  MoveL (T13144) to (117.57, 104.7, 14.9) mm, rotated rx 180 ry 0 rz -180 deg; joints [0, 0, 0, 0, 0, 0]
  Call Extruder 0.0175
  MoveL (T13145) to (117.21, 105.06, 14.9) mm, rotated rx 180 ry 0 rz -180 deg; joints [0, 0, 0, 0, 0, 0]
  Call Extruder 0.02231
  MoveL (T13146) to (117.21, 104.41, 14.9) mm, rotated rx 180 ry 0 rz -180 deg; joints [0, 0, 0, 0, 0, 0]
  Call Extruder 0.0264
  MoveL (T13147) to (117.75, 103.87, 14.9) mm, rotated rx 180 ry 0 rz -180 deg; joints [0, 0, 0, 0, 0, 0]
  Set speed (45.0 mm/s)
  Call Extruder -1.6
  MoveL (T13148) to (117.75, 103.87, 14.9) mm, rotated rx 180 ry 0 rz -180 deg; joints [0, 0, 0, 0, 0, 0]
  Set speed (120.0 mm/s)
  MoveL (T13149) to (117.75, 103.87, 14.9) mm, rotated rx 180 ry 0 rz -180 deg; joints [0, 0, 0, 0, 0, 0]
  Call Extruder -0.27367
  MoveL (T13150) to (117.21, 104.41, 14.9) mm, rotated rx 180 ry 0 rz -180 deg; joints [0, 0, 0, 0, 0, 0]
  Call Extruder -0.10633
  MoveL (T13151) to (117.21, 104.71, 14.9) mm, rotated rx 180 ry 0 rz -180 deg; joints [0, 0, 0, 0, 0, 0]
  Set speed (45.0 mm/s)
  Call Extruder -0.02
  MoveL (T13152) to (117.21, 104.71, 14.9) mm, rotated rx 180 ry 0 rz -180 deg; joints [0, 0, 0, 0, 0, 0]
  Set speed (150.0 mm/s)
  MoveL (T13153) to (117.21, 104.71, 16.9) mm, rotated rx 180 ry 0 rz -180 deg; joints [0, 0, 0, 0, 0, 0]
  MoveL (T13154) to (121.1, 106.08, 16.9) mm, rotated rx 180 ry 0 rz -180 deg; joints [0, 0, 0, 0, 0, 0]
  MoveL (T13155) to (121.1, 106.08, 14.9) mm, rotated rx 180 ry 0 rz -180 deg; joints [0, 0, 0, 0, 0, 0]
  Set speed (40.0 mm/s)
  Call Extruder 2.0
  MoveL (T13156) to (121.1, 106.08, 14.9) mm, rotated rx 180 ry 0 rz -180 deg; joints [0, 0, 0, 0, 0, 0]
  Set speed (28.1 mm/s)
  MoveL (T13157) to (121.1, 106.08, 14.9) mm, rotated rx 180 ry 0 rz -180 deg; joints [0, 0, 0, 0, 0, 0]
  Call Extruder 0.02425
  MoveL (T13158) to (120.59, 106.58, 14.9) mm, rotated rx 180 ry 0 rz -180 deg; joints [0, 0, 0, 0, 0, 0]
  Call Extruder 0.02201
  MoveL (T13159) to (119.95, 106.58, 14.9) mm, rotated rx 180 ry 0 rz -180 deg; joints [0, 0, 0, 0, 0, 0]
  Call Extruder 0.01541
  MoveL (T13160) to (120.27, 106.27, 14.9) mm, rotated rx 180 ry 0 rz -180 deg; joints [0, 0, 0, 0, 0, 0]
  Call Extruder 0.02201
  MoveL (T13161) to (119.62, 106.27, 14.9) mm, rotated rx 180 ry 0 rz -180 deg; joints [0, 0, 0, 0, 0, 0]
  Call Extruder 0.01442
  MoveL (T13162) to (119.33, 106.56, 14.9) mm, rotated rx 180 ry 0 rz -180 deg; joints [0, 0, 0, 0, 0, 0]
  Set speed (45.0 mm/s)
  Call Extruder -1.6
  MoveL (T13163) to (119.33, 106.56, 14.9) mm, rotated rx 180 ry 0 rz -180 deg; joints [0, 0, 0, 0, 0, 0]
  Set speed (120.0 mm/s)
  MoveL (T13164) to (119.33, 106.56, 14.9) mm, rotated rx 180 ry 0 rz -180 deg; joints [0, 0, 0, 0, 0, 0]
  Call Extruder -0.1506
  MoveL (T13165) to (119.62, 106.27, 14.9) mm, rotated rx 180 ry 0 rz -180 deg; joints [0, 0, 0, 0, 0, 0]
  Call Extruder -0.2294
  MoveL (T13166) to (120.27, 106.27, 14.9) mm, rotated rx 180 ry 0 rz -180 deg; joints [0, 0, 0, 0, 0, 0]
  Set speed (45.0 mm/s)
  Call Extruder -0.02
  MoveL (T13167) to (120.27, 106.27, 14.9) mm, rotated rx 180 ry 0 rz -180 deg; joints [0, 0, 0, 0, 0, 0]
  Set speed (150.0 mm/s)
  MoveL (T13168) to (120.27, 106.27, 16.9) mm, rotated rx 180 ry 0 rz -180 deg; joints [0, 0, 0, 0, 0, 0]
  MoveL (T13169) to (119.17, 110.71, 16.9) mm, rotated rx 180 ry 0 rz -180 deg; joints [0, 0, 0, 0, 0, 0]
  MoveL (T13170) to (119.17, 110.71, 14.9) mm, rotated rx 180 ry 0 rz -180 deg; joints [0, 0, 0, 0, 0, 0]
  Set speed (40.0 mm/s)
  Call Extruder 2.0
  MoveL (T13171) to (119.17, 110.71, 14.9) mm, rotated rx 180 ry 0 rz -180 deg; joints [0, 0, 0, 0, 0, 0]
  Set speed (28.1 mm/s)
  MoveL (T13172) to (119.17, 110.71, 14.9) mm, rotated rx 180 ry 0 rz -180 deg; joints [0, 0, 0, 0, 0, 0]
  Call Extruder 0.0033
  MoveL (T13173) to (119.1, 110.78, 14.9) mm, rotated rx 180 ry 0 rz -180 deg; joints [0, 0, 0, 0, 0, 0]
  Call Extruder 0.015
  MoveL (T13174) to (119.1, 111.28, 14.9) mm, rotated rx 180 ry 0 rz -180 deg; joints [0, 0, 0, 0, 0, 0]
  Call Extruder 0.01378
  MoveL (T13175) to (119.42, 111.6, 14.9) mm, rotated rx 180 ry 0 rz -180 deg; joints [0, 0, 0, 0, 0, 0]
  Call Extruder 0.04234
  MoveL (T13176) to (120.81, 111.6, 14.9) mm, rotated rx 180 ry 0 rz -180 deg; joints [0, 0, 0, 0, 0, 0]
  Call Extruder 0.01501
  MoveL (T13177) to (121.16, 111.94, 14.9) mm, rotated rx 180 ry 0 rz -180 deg; joints [0, 0, 0, 0, 0, 0]
  Call Extruder 0.01633
  MoveL (T13178) to (121.16, 112.48, 14.9) mm, rotated rx 180 ry 0 rz -180 deg; joints [0, 0, 0, 0, 0, 0]
  Call Extruder 0.05296
  MoveL (T13179) to (119.42, 112.48, 14.9) mm, rotated rx 180 ry 0 rz -180 deg; joints [0, 0, 0, 0, 0, 0]
  Call Extruder 0.00512
  MoveL (T13180) to (119.3, 112.6, 14.9) mm, rotated rx 180 ry 0 rz -180 deg; joints [0, 0, 0, 0, 0, 0]
  Set speed (150.0 mm/s)
  MoveL (T13181) to (121, 112.7, 14.9) mm, rotated rx 180 ry 0 rz -180 deg; joints [0, 0, 0, 0, 0, 0]
  Set speed (28.1 mm/s)
  MoveL (T13182) to (121, 112.7, 14.9) mm, rotated rx 180 ry 0 rz -180 deg; joints [0, 0, 0, 0, 0, 0]
  Call Extruder 0.01588
  MoveL (T13183) to (120.65, 113.05, 14.9) mm, rotated rx 180 ry 0 rz -180 deg; joints [0, 0, 0, 0, 0, 0]
  Call Extruder 0.01956
  MoveL (T13184) to (120.04, 113.05, 14.9) mm, rotated rx 180 ry 0 rz -180 deg; joints [0, 0, 0, 0, 0, 0]
  Call Extruder 0.00755
  MoveL (T13185) to (120.21, 112.89, 14.9) mm, rotated rx 180 ry 0 rz -180 deg; joints [0, 0, 0, 0, 0, 0]
  Call Extruder 0.01956
  MoveL (T13186) to (119.6, 112.89, 14.9) mm, rotated rx 180 ry 0 rz -180 deg; joints [0, 0, 0, 0, 0, 0]
  Call Extruder 0.01277
  MoveL (T13187) to (119.32, 113.17, 14.9) mm, rotated rx 180 ry 0 rz -180 deg; joints [0, 0, 0, 0, 0, 0]
  Set speed (45.0 mm/s)
  Call Extruder -1.6
  MoveL (T13188) to (119.32, 113.17, 14.9) mm, rotated rx 180 ry 0 rz -180 deg; joints [0, 0, 0, 0, 0, 0]
  Set speed (120.0 mm/s)
  MoveL (T13189) to (119.32, 113.17, 14.9) mm, rotated rx 180 ry 0 rz -180 deg; joints [0, 0, 0, 0, 0, 0]
  Call Extruder -0.14132
  MoveL (T13190) to (119.6, 112.89, 14.9) mm, rotated rx 180 ry 0 rz -180 deg; joints [0, 0, 0, 0, 0, 0]
  Call Extruder -0.21648
  MoveL (T13191) to (120.21, 112.89, 14.9) mm, rotated rx 180 ry 0 rz -180 deg; joints [0, 0, 0, 0, 0, 0]
  Call Extruder -0.0222
  MoveL (T13192) to (120.17, 112.93, 14.9) mm, rotated rx 180 ry 0 rz -180 deg; joints [0, 0, 0, 0, 0, 0]
  Set speed (45.0 mm/s)
  Call Extruder -0.02
  MoveL (T13193) to (120.17, 112.93, 14.9) mm, rotated rx 180 ry 0 rz -180 deg; joints [0, 0, 0, 0, 0, 0]
  Set speed (150.0 mm/s)
  MoveL (T13194) to (120.17, 112.93, 16.9) mm, rotated rx 180 ry 0 rz -180 deg; joints [0, 0, 0, 0, 0, 0]
  MoveL (T13195) to (120.92, 110.82, 16.9) mm, rotated rx 180 ry 0 rz -180 deg; joints [0, 0, 0, 0, 0, 0]
  MoveL (T13196) to (120.92, 110.82, 14.9) mm, rotated rx 180 ry 0 rz -180 deg; joints [0, 0, 0, 0, 0, 0]
  Set speed (40.0 mm/s)
  Call Extruder 2.0
  MoveL (T13197) to (120.92, 110.82, 14.9) mm, rotated rx 180 ry 0 rz -180 deg; joints [0, 0, 0, 0, 0, 0]
  Set speed (28.1 mm/s)
  MoveL (T13198) to (120.92, 110.82, 14.9) mm, rotated rx 180 ry 0 rz -180 deg; joints [0, 0, 0, 0, 0, 0]
  Call Extruder 0.01748
  MoveL (T13199) to (120.55, 111.19, 14.9) mm, rotated rx 180 ry 0 rz -180 deg; joints [0, 0, 0, 0, 0, 0]
  Call Extruder 0.02083
  MoveL (T13200) to (119.92, 111.19, 14.9) mm, rotated rx 180 ry 0 rz -180 deg; joints [0, 0, 0, 0, 0, 0]
  Call Extruder 0.01748
  MoveL (T13201) to (120.29, 110.82, 14.9) mm, rotated rx 180 ry 0 rz -180 deg; joints [0, 0, 0, 0, 0, 0]
  Set speed (45.0 mm/s)
  Call Extruder -1.6
  MoveL (T13202) to (120.29, 110.82, 14.9) mm, rotated rx 180 ry 0 rz -180 deg; joints [0, 0, 0, 0, 0, 0]
  Set speed (120.0 mm/s)
  MoveL (T13203) to (120.29, 110.82, 14.9) mm, rotated rx 180 ry 0 rz -180 deg; joints [0, 0, 0, 0, 0, 0]
  Call Extruder -0.18757
  MoveL (T13204) to (119.92, 111.19, 14.9) mm, rotated rx 180 ry 0 rz -180 deg; joints [0, 0, 0, 0, 0, 0]
  Call Extruder -0.19243
  MoveL (T13205) to (120.46, 111.19, 14.9) mm, rotated rx 180 ry 0 rz -180 deg; joints [0, 0, 0, 0, 0, 0]
  Set speed (45.0 mm/s)
  Call Extruder -0.02
  MoveL (T13206) to (120.46, 111.19, 14.9) mm, rotated rx 180 ry 0 rz -180 deg; joints [0, 0, 0, 0, 0, 0]
  Set speed (150.0 mm/s)
  MoveL (T13207) to (120.46, 111.19, 16.9) mm, rotated rx 180 ry 0 rz -180 deg; joints [0, 0, 0, 0, 0, 0]
  MoveL (T13208) to (121.34, 117.66, 16.9) mm, rotated rx 180 ry 0 rz -180 deg; joints [0, 0, 0, 0, 0, 0]
  MoveL (T13209) to (121.34, 117.66, 14.9) mm, rotated rx 180 ry 0 rz -180 deg; joints [0, 0, 0, 0, 0, 0]
  Set speed (40.0 mm/s)
  Call Extruder 2.0
  MoveL (T13210) to (121.34, 117.66, 14.9) mm, rotated rx 180 ry 0 rz -180 deg; joints [0, 0, 0, 0, 0, 0]
  Set speed (28.1 mm/s)
  MoveL (T13211) to (121.34, 117.66, 14.9) mm, rotated rx 180 ry 0 rz -180 deg; joints [0, 0, 0, 0, 0, 0]
  Call Extruder 0.00963
  MoveL (T13212) to (121.15, 117.85, 14.9) mm, rotated rx 180 ry 0 rz -180 deg; joints [0, 0, 0, 0, 0, 0]
  Call Extruder 0.02452
  MoveL (T13213) to (120.47, 117.85, 14.9) mm, rotated rx 180 ry 0 rz -180 deg; joints [0, 0, 0, 0, 0, 0]
  Call Extruder 0.02041
  MoveL (T13214) to (120.87, 117.45, 14.9) mm, rotated rx 180 ry 0 rz -180 deg; joints [0, 0, 0, 0, 0, 0]
  Call Extruder 0.02452
  MoveL (T13215) to (120.19, 117.45, 14.9) mm, rotated rx 180 ry 0 rz -180 deg; joints [0, 0, 0, 0, 0, 0]
  Call Extruder 0.02041
  MoveL (T13216) to (119.79, 117.85, 14.9) mm, rotated rx 180 ry 0 rz -180 deg; joints [0, 0, 0, 0, 0, 0]
  Call Extruder 0.00326
  MoveL (T13217) to (119.7, 117.85, 14.9) mm, rotated rx 180 ry 0 rz -180 deg; joints [0, 0, 0, 0, 0, 0]
  Call Extruder 0.00991
  MoveL (T13218) to (119.5, 117.65, 14.9) mm, rotated rx 180 ry 0 rz -180 deg; joints [0, 0, 0, 0, 0, 0]
  Call Extruder 0.00726
  MoveL (T13219) to (119.5, 117.45, 14.9) mm, rotated rx 180 ry 0 rz -180 deg; joints [0, 0, 0, 0, 0, 0]
  Call Extruder 0.00961
  MoveL (T13220) to (119.69, 117.26, 14.9) mm, rotated rx 180 ry 0 rz -180 deg; joints [0, 0, 0, 0, 0, 0]
  Set speed (45.0 mm/s)
  Call Extruder -1.6
  MoveL (T13221) to (119.69, 117.26, 14.9) mm, rotated rx 180 ry 0 rz -180 deg; joints [0, 0, 0, 0, 0, 0]
  Set speed (120.0 mm/s)
  MoveL (T13222) to (119.69, 117.26, 14.9) mm, rotated rx 180 ry 0 rz -180 deg; joints [0, 0, 0, 0, 0, 0]
  Call Extruder -0.09501
  MoveL (T13223) to (119.5, 117.45, 14.9) mm, rotated rx 180 ry 0 rz -180 deg; joints [0, 0, 0, 0, 0, 0]
  Call Extruder -0.07173
  MoveL (T13224) to (119.5, 117.65, 14.9) mm, rotated rx 180 ry 0 rz -180 deg; joints [0, 0, 0, 0, 0, 0]
  Call Extruder -0.09794
  MoveL (T13225) to (119.7, 117.85, 14.9) mm, rotated rx 180 ry 0 rz -180 deg; joints [0, 0, 0, 0, 0, 0]
  Call Extruder -0.03219
  MoveL (T13226) to (119.79, 117.85, 14.9) mm, rotated rx 180 ry 0 rz -180 deg; joints [0, 0, 0, 0, 0, 0]
  Call Extruder -0.08312
  MoveL (T13227) to (119.95, 117.68, 14.9) mm, rotated rx 180 ry 0 rz -180 deg; joints [0, 0, 0, 0, 0, 0]
  Set speed (45.0 mm/s)
  Call Extruder -0.02
  MoveL (T13228) to (119.95, 117.68, 14.9) mm, rotated rx 180 ry 0 rz -180 deg; joints [0, 0, 0, 0, 0, 0]
  Set speed (150.0 mm/s)
  MoveL (T13229) to (119.95, 117.68, 16.9) mm, rotated rx 180 ry 0 rz -180 deg; joints [0, 0, 0, 0, 0, 0]
  MoveL (T13230) to (104.34, 103.54, 16.9) mm, rotated rx 180 ry 0 rz -180 deg; joints [0, 0, 0, 0, 0, 0]
  MoveL (T13231) to (104.34, 103.54, 15.1) mm, rotated rx 180 ry 0 rz -180 deg; joints [0, 0, 0, 0, 0, 0]
  Set speed (40.0 mm/s)
  Call Extruder 2.0
  MoveL (T13232) to (104.34, 103.54, 15.1) mm, rotated rx 180 ry 0 rz -180 deg; joints [0, 0, 0, 0, 0, 0]
  Set speed (28.8 mm/s)
  MoveL (T13233) to (104.34, 103.54, 15.1) mm, rotated rx 180 ry 0 rz -180 deg; joints [0, 0, 0, 0, 0, 0]
  Call Extruder 0.08935
  MoveL (T13234) to (107.27, 103.54, 15.1) mm, rotated rx 180 ry 0 rz -180 deg; joints [0, 0, 0, 0, 0, 0]
  Call Extruder 0.05791
  MoveL (T13235) to (107.27, 105.44, 15.1) mm, rotated rx 180 ry 0 rz -180 deg; joints [0, 0, 0, 0, 0, 0]
  Call Extruder 0.11368
  MoveL (T13236) to (111, 105.44, 15.1) mm, rotated rx 180 ry 0 rz -180 deg; joints [0, 0, 0, 0, 0, 0]
  Call Extruder 0.05791
  MoveL (T13237) to (111, 103.54, 15.1) mm, rotated rx 180 ry 0 rz -180 deg; joints [0, 0, 0, 0, 0, 0]
  Call Extruder 0.07022
  MoveL (T13238) to (113.31, 103.54, 15.1) mm, rotated rx 180 ry 0 rz -180 deg; joints [0, 0, 0, 0, 0, 0]
  Call Extruder 0.05791
  MoveL (T13239) to (113.31, 105.44, 15.1) mm, rotated rx 180 ry 0 rz -180 deg; joints [0, 0, 0, 0, 0, 0]
  Call Extruder 0.11332
  MoveL (T13240) to (117.03, 105.44, 15.1) mm, rotated rx 180 ry 0 rz -180 deg; joints [0, 0, 0, 0, 0, 0]
  Call Extruder 0.0579
  MoveL (T13241) to (117.03, 103.54, 15.1) mm, rotated rx 180 ry 0 rz -180 deg; joints [0, 0, 0, 0, 0, 0]
  Call Extruder 0.13501
  MoveL (T13242) to (121.46, 103.54, 15.1) mm, rotated rx 180 ry 0 rz -180 deg; joints [0, 0, 0, 0, 0, 0]
  Call Extruder 0.09842
  MoveL (T13243) to (121.46, 106.77, 15.1) mm, rotated rx 180 ry 0 rz -180 deg; joints [0, 0, 0, 0, 0, 0]
  Call Extruder 0.05868
  MoveL (T13244) to (119.53, 106.77, 15.1) mm, rotated rx 180 ry 0 rz -180 deg; joints [0, 0, 0, 0, 0, 0]
  Call Extruder 0.11599
  MoveL (T13245) to (119.53, 110.58, 15.1) mm, rotated rx 180 ry 0 rz -180 deg; joints [0, 0, 0, 0, 0, 0]
  Call Extruder 0.05873
  MoveL (T13246) to (121.46, 110.58, 15.1) mm, rotated rx 180 ry 0 rz -180 deg; joints [0, 0, 0, 0, 0, 0]
  Call Extruder 0.08813
  MoveL (T13247) to (121.46, 113.47, 15.1) mm, rotated rx 180 ry 0 rz -180 deg; joints [0, 0, 0, 0, 0, 0]
  Call Extruder 0.05877
  MoveL (T13248) to (119.53, 113.47, 15.1) mm, rotated rx 180 ry 0 rz -180 deg; joints [0, 0, 0, 0, 0, 0]
  Call Extruder 0.11538
  MoveL (T13249) to (119.53, 117.25, 15.1) mm, rotated rx 180 ry 0 rz -180 deg; joints [0, 0, 0, 0, 0, 0]
  Call Extruder 0.05882
  MoveL (T13250) to (121.46, 117.26, 15.1) mm, rotated rx 180 ry 0 rz -180 deg; joints [0, 0, 0, 0, 0, 0]
  Call Extruder 0.12804
  MoveL (T13251) to (121.46, 121.46, 15.1) mm, rotated rx 180 ry 0 rz -180 deg; joints [0, 0, 0, 0, 0, 0]
  Call Extruder 0.54596
  MoveL (T13252) to (103.54, 121.46, 15.1) mm, rotated rx 180 ry 0 rz -180 deg; joints [0, 0, 0, 0, 0, 0]
  Call Extruder 0.54596
  MoveL (T13253) to (103.54, 103.54, 15.1) mm, rotated rx 180 ry 0 rz -180 deg; joints [0, 0, 0, 0, 0, 0]
  Call Extruder 0.02254
  MoveL (T13254) to (104.28, 103.54, 15.1) mm, rotated rx 180 ry 0 rz -180 deg; joints [0, 0, 0, 0, 0, 0]
  Set speed (150.0 mm/s)
  MoveL (T13255) to (103.53, 103.13, 15.1) mm, rotated rx 180 ry 0 rz -180 deg; joints [0, 0, 0, 0, 0, 0]
  Set speed (28.8 mm/s)
  MoveL (T13256) to (103.53, 103.13, 15.1) mm, rotated rx 180 ry 0 rz -180 deg; joints [0, 0, 0, 0, 0, 0]
  Call Extruder 0.12635
  MoveL (T13257) to (107.68, 103.13, 15.1) mm, rotated rx 180 ry 0 rz -180 deg; joints [0, 0, 0, 0, 0, 0]
  Call Extruder 0.05791
  MoveL (T13258) to (107.68, 105.03, 15.1) mm, rotated rx 180 ry 0 rz -180 deg; joints [0, 0, 0, 0, 0, 0]
  Call Extruder 0.08888
  MoveL (T13259) to (110.6, 105.03, 15.1) mm, rotated rx 180 ry 0 rz -180 deg; joints [0, 0, 0, 0, 0, 0]
  Call Extruder 0.05791
  MoveL (T13260) to (110.6, 103.13, 15.1) mm, rotated rx 180 ry 0 rz -180 deg; joints [0, 0, 0, 0, 0, 0]
  Call Extruder 0.09501
  MoveL (T13261) to (113.72, 103.13, 15.1) mm, rotated rx 180 ry 0 rz -180 deg; joints [0, 0, 0, 0, 0, 0]
  Call Extruder 0.05791
  MoveL (T13262) to (113.72, 105.03, 15.1) mm, rotated rx 180 ry 0 rz -180 deg; joints [0, 0, 0, 0, 0, 0]
  Call Extruder 0.08852
  MoveL (T13263) to (116.62, 105.03, 15.1) mm, rotated rx 180 ry 0 rz -180 deg; joints [0, 0, 0, 0, 0, 0]
  Call Extruder 0.0579
  MoveL (T13264) to (116.62, 103.13, 15.1) mm, rotated rx 180 ry 0 rz -180 deg; joints [0, 0, 0, 0, 0, 0]
  Call Extruder 0.15982
  MoveL (T13265) to (121.87, 103.13, 15.1) mm, rotated rx 180 ry 0 rz -180 deg; joints [0, 0, 0, 0, 0, 0]
  Call Extruder 0.12322
  MoveL (T13266) to (121.87, 107.18, 15.1) mm, rotated rx 180 ry 0 rz -180 deg; joints [0, 0, 0, 0, 0, 0]
  Call Extruder 0.05868
  MoveL (T13267) to (119.94, 107.18, 15.1) mm, rotated rx 180 ry 0 rz -180 deg; joints [0, 0, 0, 0, 0, 0]
  Call Extruder 0.09119
  MoveL (T13268) to (119.94, 110.17, 15.1) mm, rotated rx 180 ry 0 rz -180 deg; joints [0, 0, 0, 0, 0, 0]
  Call Extruder 0.05872
  MoveL (T13269) to (121.87, 110.17, 15.1) mm, rotated rx 180 ry 0 rz -180 deg; joints [0, 0, 0, 0, 0, 0]
  Call Extruder 0.11295
  MoveL (T13270) to (121.87, 113.88, 15.1) mm, rotated rx 180 ry 0 rz -180 deg; joints [0, 0, 0, 0, 0, 0]
  Call Extruder 0.05877
  MoveL (T13271) to (119.94, 113.88, 15.1) mm, rotated rx 180 ry 0 rz -180 deg; joints [0, 0, 0, 0, 0, 0]
  Call Extruder 0.09058
  MoveL (T13272) to (119.94, 116.85, 15.1) mm, rotated rx 180 ry 0 rz -180 deg; joints [0, 0, 0, 0, 0, 0]
  Call Extruder 0.05881
  MoveL (T13273) to (121.87, 116.85, 15.1) mm, rotated rx 180 ry 0 rz -180 deg; joints [0, 0, 0, 0, 0, 0]
  Call Extruder 0.15282
  MoveL (T13274) to (121.87, 121.87, 15.1) mm, rotated rx 180 ry 0 rz -180 deg; joints [0, 0, 0, 0, 0, 0]
  Call Extruder 0.57077
  MoveL (T13275) to (103.13, 121.87, 15.1) mm, rotated rx 180 ry 0 rz -180 deg; joints [0, 0, 0, 0, 0, 0]
  Call Extruder 0.57077
  MoveL (T13276) to (103.13, 103.13, 15.1) mm, rotated rx 180 ry 0 rz -180 deg; joints [0, 0, 0, 0, 0, 0]
  Call Extruder 0.01036
  MoveL (T13277) to (103.47, 103.13, 15.1) mm, rotated rx 180 ry 0 rz -180 deg; joints [0, 0, 0, 0, 0, 0]
  Set speed (150.0 mm/s)
  MoveL (T13278) to (102.72, 102.81, 15.1) mm, rotated rx 180 ry 0 rz -180 deg; joints [0, 0, 0, 0, 0, 0]
  Set speed (25.0 mm/s)
  MoveL (T13279) to (102.72, 102.81, 15.1) mm, rotated rx 180 ry 0 rz -180 deg; joints [0, 0, 0, 0, 0, 0]
  Call Extruder 0.00259
  MoveL (T13280) to (102.72, 102.72, 15.1) mm, rotated rx 180 ry 0 rz -180 deg; joints [0, 0, 0, 0, 0, 0]
  Call Extruder 0.16334
  MoveL (T13281) to (108.09, 102.72, 15.1) mm, rotated rx 180 ry 0 rz -180 deg; joints [0, 0, 0, 0, 0, 0]
  Call Extruder 0.05791
  MoveL (T13282) to (108.09, 104.63, 15.1) mm, rotated rx 180 ry 0 rz -180 deg; joints [0, 0, 0, 0, 0, 0]
  Call Extruder 0.06408
  MoveL (T13283) to (110.19, 104.63, 15.1) mm, rotated rx 180 ry 0 rz -180 deg; joints [0, 0, 0, 0, 0, 0]
  Call Extruder 0.05791
  MoveL (T13284) to (110.19, 102.72, 15.1) mm, rotated rx 180 ry 0 rz -180 deg; joints [0, 0, 0, 0, 0, 0]
  Call Extruder 0.1198
  MoveL (T13285) to (114.12, 102.72, 15.1) mm, rotated rx 180 ry 0 rz -180 deg; joints [0, 0, 0, 0, 0, 0]
  Call Extruder 0.05791
  MoveL (T13286) to (114.12, 104.63, 15.1) mm, rotated rx 180 ry 0 rz -180 deg; joints [0, 0, 0, 0, 0, 0]
  Call Extruder 0.06372
  MoveL (T13287) to (116.22, 104.63, 15.1) mm, rotated rx 180 ry 0 rz -180 deg; joints [0, 0, 0, 0, 0, 0]
  Call Extruder 0.0579
  MoveL (T13288) to (116.21, 102.72, 15.1) mm, rotated rx 180 ry 0 rz -180 deg; joints [0, 0, 0, 0, 0, 0]
  Call Extruder 0.18463
  MoveL (T13289) to (122.28, 102.72, 15.1) mm, rotated rx 180 ry 0 rz -180 deg; joints [0, 0, 0, 0, 0, 0]
  Call Extruder 0.14802
  MoveL (T13290) to (122.28, 107.58, 15.1) mm, rotated rx 180 ry 0 rz -180 deg; joints [0, 0, 0, 0, 0, 0]
  Call Extruder 0.05869
  MoveL (T13291) to (120.35, 107.58, 15.1) mm, rotated rx 180 ry 0 rz -180 deg; joints [0, 0, 0, 0, 0, 0]
  Call Extruder 0.06638
  MoveL (T13292) to (120.35, 109.76, 15.1) mm, rotated rx 180 ry 0 rz -180 deg; joints [0, 0, 0, 0, 0, 0]
  Call Extruder 0.05872
  MoveL (T13293) to (122.28, 109.76, 15.1) mm, rotated rx 180 ry 0 rz -180 deg; joints [0, 0, 0, 0, 0, 0]
  Call Extruder 0.13778
  MoveL (T13294) to (122.28, 114.29, 15.1) mm, rotated rx 180 ry 0 rz -180 deg; joints [0, 0, 0, 0, 0, 0]
  Call Extruder 0.05878
  MoveL (T13295) to (120.35, 114.28, 15.1) mm, rotated rx 180 ry 0 rz -180 deg; joints [0, 0, 0, 0, 0, 0]
  Call Extruder 0.06578
  MoveL (T13296) to (120.34, 116.44, 15.1) mm, rotated rx 180 ry 0 rz -180 deg; joints [0, 0, 0, 0, 0, 0]
  Call Extruder 0.05881
  MoveL (T13297) to (122.28, 116.44, 15.1) mm, rotated rx 180 ry 0 rz -180 deg; joints [0, 0, 0, 0, 0, 0]
  Call Extruder 0.17761
  MoveL (T13298) to (122.28, 122.28, 15.1) mm, rotated rx 180 ry 0 rz -180 deg; joints [0, 0, 0, 0, 0, 0]
  Call Extruder 0.59557
  MoveL (T13299) to (102.72, 122.28, 15.1) mm, rotated rx 180 ry 0 rz -180 deg; joints [0, 0, 0, 0, 0, 0]
  Call Extruder 0.59115
  MoveL (T13300) to (102.72, 102.87, 15.1) mm, rotated rx 180 ry 0 rz -180 deg; joints [0, 0, 0, 0, 0, 0]
  Set speed (150.0 mm/s)
  MoveL (T13301) to (102.78, 102.75, 15.1) mm, rotated rx 180 ry 0 rz -180 deg; joints [0, 0, 0, 0, 0, 0]
  Set speed (45.0 mm/s)
  Call Extruder -1.6
  MoveL (T13302) to (102.78, 102.75, 15.1) mm, rotated rx 180 ry 0 rz -180 deg; joints [0, 0, 0, 0, 0, 0]
  Set speed (120.0 mm/s)
  MoveL (T13303) to (102.78, 102.75, 15.1) mm, rotated rx 180 ry 0 rz -180 deg; joints [0, 0, 0, 0, 0, 0]
  Call Extruder -0.05166
  MoveL (T13304) to (102.72, 102.72, 15.1) mm, rotated rx 180 ry 0 rz -180 deg; joints [0, 0, 0, 0, 0, 0]
  Call Extruder -0.32834
  MoveL (T13305) to (103.65, 102.72, 15.1) mm, rotated rx 180 ry 0 rz -180 deg; joints [0, 0, 0, 0, 0, 0]
  Set speed (45.0 mm/s)
  Call Extruder -0.02
  MoveL (T13306) to (103.65, 102.72, 15.1) mm, rotated rx 180 ry 0 rz -180 deg; joints [0, 0, 0, 0, 0, 0]
  Set speed (150.0 mm/s)
  MoveL (T13307) to (103.65, 102.72, 17.1) mm, rotated rx 180 ry 0 rz -180 deg; joints [0, 0, 0, 0, 0, 0]
  MoveL (T13308) to (106.29, 103.84, 17.1) mm, rotated rx 180 ry 0 rz -180 deg; joints [0, 0, 0, 0, 0, 0]
  MoveL (T13309) to (106.29, 103.84, 15.1) mm, rotated rx 180 ry 0 rz -180 deg; joints [0, 0, 0, 0, 0, 0]
  Set speed (40.0 mm/s)
  Call Extruder 2.0
  MoveL (T13310) to (106.29, 103.84, 15.1) mm, rotated rx 180 ry 0 rz -180 deg; joints [0, 0, 0, 0, 0, 0]
  Set speed (28.8 mm/s)
  MoveL (T13311) to (106.29, 103.84, 15.1) mm, rotated rx 180 ry 0 rz -180 deg; joints [0, 0, 0, 0, 0, 0]
  Call Extruder 0.07441
  MoveL (T13312) to (103.84, 103.84, 15.1) mm, rotated rx 180 ry 0 rz -180 deg; joints [0, 0, 0, 0, 0, 0]
  Call Extruder 0.7458
  MoveL (T13313) to (121.16, 121.16, 15.1) mm, rotated rx 180 ry 0 rz -180 deg; joints [0, 0, 0, 0, 0, 0]
  Call Extruder 0.08828
  MoveL (T13314) to (121.16, 118.26, 15.1) mm, rotated rx 180 ry 0 rz -180 deg; joints [0, 0, 0, 0, 0, 0]
  Call Extruder 0.01815
  MoveL (T13315) to (120.56, 118.26, 15.1) mm, rotated rx 180 ry 0 rz -180 deg; joints [0, 0, 0, 0, 0, 0]
  Call Extruder 0.12488
  MoveL (T13316) to (117.66, 121.16, 15.1) mm, rotated rx 180 ry 0 rz -180 deg; joints [0, 0, 0, 0, 0, 0]
  Call Extruder 0.03385
  MoveL (T13317) to (116.55, 121.16, 15.1) mm, rotated rx 180 ry 0 rz -180 deg; joints [0, 0, 0, 0, 0, 0]
  Call Extruder 0.54738
  MoveL (T13318) to (103.84, 108.45, 15.1) mm, rotated rx 180 ry 0 rz -180 deg; joints [0, 0, 0, 0, 0, 0]
  Call Extruder 0.03385
  MoveL (T13319) to (103.84, 107.34, 15.1) mm, rotated rx 180 ry 0 rz -180 deg; joints [0, 0, 0, 0, 0, 0]
  Call Extruder 0.10959
  MoveL (T13320) to (106.39, 104.8, 15.1) mm, rotated rx 180 ry 0 rz -180 deg; joints [0, 0, 0, 0, 0, 0]
  Call Extruder 0.02313
  MoveL (T13321) to (106.39, 105.55, 15.1) mm, rotated rx 180 ry 0 rz -180 deg; joints [0, 0, 0, 0, 0, 0]
  Call Extruder 0.01377
  MoveL (T13322) to (106.71, 105.87, 15.1) mm, rotated rx 180 ry 0 rz -180 deg; joints [0, 0, 0, 0, 0, 0]
  Call Extruder 0.01445
  MoveL (T13323) to (107.18, 105.87, 15.1) mm, rotated rx 180 ry 0 rz -180 deg; joints [0, 0, 0, 0, 0, 0]
  Call Extruder 0.00555
  MoveL (T13324) to (107.31, 105.75, 15.1) mm, rotated rx 180 ry 0 rz -180 deg; joints [0, 0, 0, 0, 0, 0]
  Call Extruder 0.0175
  MoveL (T13325) to (107.89, 105.75, 15.1) mm, rotated rx 180 ry 0 rz -180 deg; joints [0, 0, 0, 0, 0, 0]
  Set speed (45.0 mm/s)
  Call Extruder -1.6
  MoveL (T13326) to (107.89, 105.75, 15.1) mm, rotated rx 180 ry 0 rz -180 deg; joints [0, 0, 0, 0, 0, 0]
  Set speed (120.0 mm/s)
  MoveL (T13327) to (107.89, 105.75, 15.1) mm, rotated rx 180 ry 0 rz -180 deg; joints [0, 0, 0, 0, 0, 0]
  Call Extruder -0.2046
  MoveL (T13328) to (107.31, 105.75, 15.1) mm, rotated rx 180 ry 0 rz -180 deg; joints [0, 0, 0, 0, 0, 0]
  Call Extruder -0.06495
  MoveL (T13329) to (107.18, 105.87, 15.1) mm, rotated rx 180 ry 0 rz -180 deg; joints [0, 0, 0, 0, 0, 0]
  Call Extruder -0.11045
  MoveL (T13330) to (106.87, 105.87, 15.1) mm, rotated rx 180 ry 0 rz -180 deg; joints [0, 0, 0, 0, 0, 0]
  Set speed (45.0 mm/s)
  Call Extruder -0.02
  MoveL (T13331) to (106.87, 105.87, 15.1) mm, rotated rx 180 ry 0 rz -180 deg; joints [0, 0, 0, 0, 0, 0]
  Set speed (150.0 mm/s)
  MoveL (T13332) to (106.87, 105.87, 17.1) mm, rotated rx 180 ry 0 rz -180 deg; joints [0, 0, 0, 0, 0, 0]
  MoveL (T13333) to (106.61, 103.99, 17.1) mm, rotated rx 180 ry 0 rz -180 deg; joints [0, 0, 0, 0, 0, 0]
  MoveL (T13334) to (106.61, 103.99, 15.1) mm, rotated rx 180 ry 0 rz -180 deg; joints [0, 0, 0, 0, 0, 0]
  Set speed (40.0 mm/s)
  Call Extruder 2.0
  MoveL (T13335) to (106.61, 103.99, 15.1) mm, rotated rx 180 ry 0 rz -180 deg; joints [0, 0, 0, 0, 0, 0]
  Set speed (28.8 mm/s)
  MoveL (T13336) to (106.61, 103.99, 15.1) mm, rotated rx 180 ry 0 rz -180 deg; joints [0, 0, 0, 0, 0, 0]
  Call Extruder 0.01595
  MoveL (T13337) to (106.97, 104.34, 15.1) mm, rotated rx 180 ry 0 rz -180 deg; joints [0, 0, 0, 0, 0, 0]
  Call Extruder 0.01917
  MoveL (T13338) to (106.97, 104.94, 15.1) mm, rotated rx 180 ry 0 rz -180 deg; joints [0, 0, 0, 0, 0, 0]
  Call Extruder 0.0077
  MoveL (T13339) to (106.8, 104.77, 15.1) mm, rotated rx 180 ry 0 rz -180 deg; joints [0, 0, 0, 0, 0, 0]
  Call Extruder 0.01917
  MoveL (T13340) to (106.8, 105.37, 15.1) mm, rotated rx 180 ry 0 rz -180 deg; joints [0, 0, 0, 0, 0, 0]
  Call Extruder 0.0125
  MoveL (T13341) to (107.07, 105.65, 15.1) mm, rotated rx 180 ry 0 rz -180 deg; joints [0, 0, 0, 0, 0, 0]
  Set speed (45.0 mm/s)
  Call Extruder -1.6
  MoveL (T13342) to (107.07, 105.65, 15.1) mm, rotated rx 180 ry 0 rz -180 deg; joints [0, 0, 0, 0, 0, 0]
  Set speed (120.0 mm/s)
  MoveL (T13343) to (107.07, 105.65, 15.1) mm, rotated rx 180 ry 0 rz -180 deg; joints [0, 0, 0, 0, 0, 0]
  Call Extruder -0.13974
  MoveL (T13344) to (106.8, 105.37, 15.1) mm, rotated rx 180 ry 0 rz -180 deg; joints [0, 0, 0, 0, 0, 0]
  Call Extruder -0.21439
  MoveL (T13345) to (106.8, 104.77, 15.1) mm, rotated rx 180 ry 0 rz -180 deg; joints [0, 0, 0, 0, 0, 0]
  Call Extruder -0.02587
  MoveL (T13346) to (106.85, 104.82, 15.1) mm, rotated rx 180 ry 0 rz -180 deg; joints [0, 0, 0, 0, 0, 0]
  Set speed (45.0 mm/s)
  Call Extruder -0.02
  MoveL (T13347) to (106.85, 104.82, 15.1) mm, rotated rx 180 ry 0 rz -180 deg; joints [0, 0, 0, 0, 0, 0]
  Set speed (150.0 mm/s)
  MoveL (T13348) to (106.85, 104.82, 17.1) mm, rotated rx 180 ry 0 rz -180 deg; joints [0, 0, 0, 0, 0, 0]
  MoveL (T13349) to (111.23, 105.87, 17.1) mm, rotated rx 180 ry 0 rz -180 deg; joints [0, 0, 0, 0, 0, 0]
  MoveL (T13350) to (111.23, 105.87, 15.1) mm, rotated rx 180 ry 0 rz -180 deg; joints [0, 0, 0, 0, 0, 0]
  Set speed (40.0 mm/s)
  Call Extruder 2.0
  MoveL (T13351) to (111.23, 105.87, 15.1) mm, rotated rx 180 ry 0 rz -180 deg; joints [0, 0, 0, 0, 0, 0]
  Set speed (28.8 mm/s)
  MoveL (T13352) to (111.23, 105.87, 15.1) mm, rotated rx 180 ry 0 rz -180 deg; joints [0, 0, 0, 0, 0, 0]
  Call Extruder 0.01028
  MoveL (T13353) to (111.57, 105.87, 15.1) mm, rotated rx 180 ry 0 rz -180 deg; joints [0, 0, 0, 0, 0, 0]
  Call Extruder 0.01375
  MoveL (T13354) to (111.89, 105.55, 15.1) mm, rotated rx 180 ry 0 rz -180 deg; joints [0, 0, 0, 0, 0, 0]
  Call Extruder 0.05038
  MoveL (T13355) to (111.89, 103.9, 15.1) mm, rotated rx 180 ry 0 rz -180 deg; joints [0, 0, 0, 0, 0, 0]
  Call Extruder 0.00237
  MoveL (T13356) to (111.94, 103.84, 15.1) mm, rotated rx 180 ry 0 rz -180 deg; joints [0, 0, 0, 0, 0, 0]
  Call Extruder 0.01299
  MoveL (T13357) to (112.37, 103.84, 15.1) mm, rotated rx 180 ry 0 rz -180 deg; joints [0, 0, 0, 0, 0, 0]
  Call Extruder 0.05207
  MoveL (T13358) to (112.37, 105.55, 15.1) mm, rotated rx 180 ry 0 rz -180 deg; joints [0, 0, 0, 0, 0, 0]
  Call Extruder 0.00935
  MoveL (T13359) to (112.59, 105.77, 15.1) mm, rotated rx 180 ry 0 rz -180 deg; joints [0, 0, 0, 0, 0, 0]
  Set speed (150.0 mm/s)
  MoveL (T13360) to (112.59, 103.95, 15.1) mm, rotated rx 180 ry 0 rz -180 deg; joints [0, 0, 0, 0, 0, 0]
  Set speed (28.8 mm/s)
  MoveL (T13361) to (112.59, 103.95, 15.1) mm, rotated rx 180 ry 0 rz -180 deg; joints [0, 0, 0, 0, 0, 0]
  Call Extruder 0.01886
  MoveL (T13362) to (113, 104.36, 15.1) mm, rotated rx 180 ry 0 rz -180 deg; joints [0, 0, 0, 0, 0, 0]
  Call Extruder 0.02004
  MoveL (T13363) to (113, 104.98, 15.1) mm, rotated rx 180 ry 0 rz -180 deg; joints [0, 0, 0, 0, 0, 0]
  Call Extruder 0.01042
  MoveL (T13364) to (112.78, 104.75, 15.1) mm, rotated rx 180 ry 0 rz -180 deg; joints [0, 0, 0, 0, 0, 0]
  Call Extruder 0.02004
  MoveL (T13365) to (112.78, 105.36, 15.1) mm, rotated rx 180 ry 0 rz -180 deg; joints [0, 0, 0, 0, 0, 0]
  Call Extruder 0.01308
  MoveL (T13366) to (113.06, 105.65, 15.1) mm, rotated rx 180 ry 0 rz -180 deg; joints [0, 0, 0, 0, 0, 0]
  Set speed (45.0 mm/s)
  Call Extruder -1.6
  MoveL (T13367) to (113.06, 105.65, 15.1) mm, rotated rx 180 ry 0 rz -180 deg; joints [0, 0, 0, 0, 0, 0]
  Set speed (120.0 mm/s)
  MoveL (T13368) to (113.06, 105.65, 15.1) mm, rotated rx 180 ry 0 rz -180 deg; joints [0, 0, 0, 0, 0, 0]
  Call Extruder -0.1431
  MoveL (T13369) to (112.78, 105.36, 15.1) mm, rotated rx 180 ry 0 rz -180 deg; joints [0, 0, 0, 0, 0, 0]
  Call Extruder -0.21928
  MoveL (T13370) to (112.78, 104.75, 15.1) mm, rotated rx 180 ry 0 rz -180 deg; joints [0, 0, 0, 0, 0, 0]
  Call Extruder -0.01762
  MoveL (T13371) to (112.81, 104.78, 15.1) mm, rotated rx 180 ry 0 rz -180 deg; joints [0, 0, 0, 0, 0, 0]
  Set speed (45.0 mm/s)
  Call Extruder -0.02
  MoveL (T13372) to (112.81, 104.78, 15.1) mm, rotated rx 180 ry 0 rz -180 deg; joints [0, 0, 0, 0, 0, 0]
  Set speed (150.0 mm/s)
  MoveL (T13373) to (112.81, 104.78, 17.1) mm, rotated rx 180 ry 0 rz -180 deg; joints [0, 0, 0, 0, 0, 0]
  MoveL (T13374) to (111.13, 104.08, 17.1) mm, rotated rx 180 ry 0 rz -180 deg; joints [0, 0, 0, 0, 0, 0]
  MoveL (T13375) to (111.13, 104.08, 15.1) mm, rotated rx 180 ry 0 rz -180 deg; joints [0, 0, 0, 0, 0, 0]
  Set speed (40.0 mm/s)
  Call Extruder 2.0
  MoveL (T13376) to (111.13, 104.08, 15.1) mm, rotated rx 180 ry 0 rz -180 deg; joints [0, 0, 0, 0, 0, 0]
  Set speed (28.8 mm/s)
  MoveL (T13377) to (111.13, 104.08, 15.1) mm, rotated rx 180 ry 0 rz -180 deg; joints [0, 0, 0, 0, 0, 0]
  Call Extruder 0.01643
  MoveL (T13378) to (111.48, 104.43, 15.1) mm, rotated rx 180 ry 0 rz -180 deg; joints [0, 0, 0, 0, 0, 0]
  Call Extruder 0.02009
  MoveL (T13379) to (111.48, 105.05, 15.1) mm, rotated rx 180 ry 0 rz -180 deg; joints [0, 0, 0, 0, 0, 0]
  Call Extruder 0.01643
  MoveL (T13380) to (111.13, 104.69, 15.1) mm, rotated rx 180 ry 0 rz -180 deg; joints [0, 0, 0, 0, 0, 0]
  Set speed (45.0 mm/s)
  Call Extruder -1.6
  MoveL (T13381) to (111.13, 104.69, 15.1) mm, rotated rx 180 ry 0 rz -180 deg; joints [0, 0, 0, 0, 0, 0]
  Set speed (120.0 mm/s)
  MoveL (T13382) to (111.13, 104.69, 15.1) mm, rotated rx 180 ry 0 rz -180 deg; joints [0, 0, 0, 0, 0, 0]
  Call Extruder -0.17945
  MoveL (T13383) to (111.48, 105.05, 15.1) mm, rotated rx 180 ry 0 rz -180 deg; joints [0, 0, 0, 0, 0, 0]
  Call Extruder -0.20055
  MoveL (T13384) to (111.48, 104.49, 15.1) mm, rotated rx 180 ry 0 rz -180 deg; joints [0, 0, 0, 0, 0, 0]
  Set speed (45.0 mm/s)
  Call Extruder -0.02
  MoveL (T13385) to (111.48, 104.49, 15.1) mm, rotated rx 180 ry 0 rz -180 deg; joints [0, 0, 0, 0, 0, 0]
  Set speed (150.0 mm/s)
  MoveL (T13386) to (111.48, 104.49, 17.1) mm, rotated rx 180 ry 0 rz -180 deg; joints [0, 0, 0, 0, 0, 0]
  MoveL (T13387) to (117.15, 104.04, 17.1) mm, rotated rx 180 ry 0 rz -180 deg; joints [0, 0, 0, 0, 0, 0]
  MoveL (T13388) to (117.15, 104.04, 15.1) mm, rotated rx 180 ry 0 rz -180 deg; joints [0, 0, 0, 0, 0, 0]
  Set speed (40.0 mm/s)
  Call Extruder 2.0
  MoveL (T13389) to (117.15, 104.04, 15.1) mm, rotated rx 180 ry 0 rz -180 deg; joints [0, 0, 0, 0, 0, 0]
  Set speed (28.8 mm/s)
  MoveL (T13390) to (117.15, 104.04, 15.1) mm, rotated rx 180 ry 0 rz -180 deg; joints [0, 0, 0, 0, 0, 0]
  Call Extruder 0.01964
  MoveL (T13391) to (117.57, 104.46, 15.1) mm, rotated rx 180 ry 0 rz -180 deg; joints [0, 0, 0, 0, 0, 0]
  Call Extruder 0.02109
  MoveL (T13392) to (117.57, 105.09, 15.1) mm, rotated rx 180 ry 0 rz -180 deg; joints [0, 0, 0, 0, 0, 0]
  Call Extruder 0.01964
  MoveL (T13393) to (117.15, 104.67, 15.1) mm, rotated rx 180 ry 0 rz -180 deg; joints [0, 0, 0, 0, 0, 0]
  Set speed (150.0 mm/s)
  MoveL (T13394) to (117.08, 105.83, 15.1) mm, rotated rx 180 ry 0 rz -180 deg; joints [0, 0, 0, 0, 0, 0]
  Set speed (28.8 mm/s)
  MoveL (T13395) to (117.08, 105.83, 15.1) mm, rotated rx 180 ry 0 rz -180 deg; joints [0, 0, 0, 0, 0, 0]
  Call Extruder 0.00176
  MoveL (T13396) to (117.12, 105.87, 15.1) mm, rotated rx 180 ry 0 rz -180 deg; joints [0, 0, 0, 0, 0, 0]
  Call Extruder 0.01632
  MoveL (T13397) to (117.66, 105.87, 15.1) mm, rotated rx 180 ry 0 rz -180 deg; joints [0, 0, 0, 0, 0, 0]
  Call Extruder 0.01377
  MoveL (T13398) to (117.97, 105.55, 15.1) mm, rotated rx 180 ry 0 rz -180 deg; joints [0, 0, 0, 0, 0, 0]
  Call Extruder 0.04255
  MoveL (T13399) to (117.97, 104.16, 15.1) mm, rotated rx 180 ry 0 rz -180 deg; joints [0, 0, 0, 0, 0, 0]
  Call Extruder 0.0733
  MoveL (T13400) to (119.68, 105.86, 15.1) mm, rotated rx 180 ry 0 rz -180 deg; joints [0, 0, 0, 0, 0, 0]
  Call Extruder 0.04508
  MoveL (T13401) to (121.16, 105.86, 15.1) mm, rotated rx 180 ry 0 rz -180 deg; joints [0, 0, 0, 0, 0, 0]
  Call Extruder 0.06135
  MoveL (T13402) to (121.16, 103.84, 15.1) mm, rotated rx 180 ry 0 rz -180 deg; joints [0, 0, 0, 0, 0, 0]
  Call Extruder 0.7458
  MoveL (T13403) to (103.84, 121.16, 15.1) mm, rotated rx 180 ry 0 rz -180 deg; joints [0, 0, 0, 0, 0, 0]
  Call Extruder 0.10645
  MoveL (T13404) to (103.84, 117.66, 15.1) mm, rotated rx 180 ry 0 rz -180 deg; joints [0, 0, 0, 0, 0, 0]
  Call Extruder 0.15054
  MoveL (T13405) to (107.34, 121.16, 15.1) mm, rotated rx 180 ry 0 rz -180 deg; joints [0, 0, 0, 0, 0, 0]
  Call Extruder 0.03385
  MoveL (T13406) to (108.45, 121.16, 15.1) mm, rotated rx 180 ry 0 rz -180 deg; joints [0, 0, 0, 0, 0, 0]
  Call Extruder 0.46434
  MoveL (T13407) to (119.23, 110.38, 15.1) mm, rotated rx 180 ry 0 rz -180 deg; joints [0, 0, 0, 0, 0, 0]
  Call Extruder 0.01099
  MoveL (T13408) to (119.23, 110.02, 15.1) mm, rotated rx 180 ry 0 rz -180 deg; joints [0, 0, 0, 0, 0, 0]
  Call Extruder 0.18403
  MoveL (T13409) to (114.96, 105.75, 15.1) mm, rotated rx 180 ry 0 rz -180 deg; joints [0, 0, 0, 0, 0, 0]
  Call Extruder 0.00936
  MoveL (T13410) to (114.65, 105.75, 15.1) mm, rotated rx 180 ry 0 rz -180 deg; joints [0, 0, 0, 0, 0, 0]
  Call Extruder 0.46549
  MoveL (T13411) to (103.84, 116.55, 15.1) mm, rotated rx 180 ry 0 rz -180 deg; joints [0, 0, 0, 0, 0, 0]
  Call Extruder 0.10645
  MoveL (T13412) to (103.84, 113.06, 15.1) mm, rotated rx 180 ry 0 rz -180 deg; joints [0, 0, 0, 0, 0, 0]
  Call Extruder 0.34896
  MoveL (T13413) to (111.94, 121.16, 15.1) mm, rotated rx 180 ry 0 rz -180 deg; joints [0, 0, 0, 0, 0, 0]
  Call Extruder 0.03385
  MoveL (T13414) to (113.06, 121.16, 15.1) mm, rotated rx 180 ry 0 rz -180 deg; joints [0, 0, 0, 0, 0, 0]
  Call Extruder 0.26583
  MoveL (T13415) to (119.23, 114.98, 15.1) mm, rotated rx 180 ry 0 rz -180 deg; joints [0, 0, 0, 0, 0, 0]
  Call Extruder 0.01112
  MoveL (T13416) to (119.23, 114.62, 15.1) mm, rotated rx 180 ry 0 rz -180 deg; joints [0, 0, 0, 0, 0, 0]
  Call Extruder 0.38236
  MoveL (T13417) to (110.35, 105.75, 15.1) mm, rotated rx 180 ry 0 rz -180 deg; joints [0, 0, 0, 0, 0, 0]
  Call Extruder 0.00936
  MoveL (T13418) to (110.04, 105.75, 15.1) mm, rotated rx 180 ry 0 rz -180 deg; joints [0, 0, 0, 0, 0, 0]
  Call Extruder 0.26707
  MoveL (T13419) to (103.84, 111.94, 15.1) mm, rotated rx 180 ry 0 rz -180 deg; joints [0, 0, 0, 0, 0, 0]
  Call Extruder 0.07441
  MoveL (T13420) to (103.84, 109.5, 15.1) mm, rotated rx 180 ry 0 rz -180 deg; joints [0, 0, 0, 0, 0, 0]
  Set speed (45.0 mm/s)
  Call Extruder -1.6
  MoveL (T13421) to (103.84, 109.5, 15.1) mm, rotated rx 180 ry 0 rz -180 deg; joints [0, 0, 0, 0, 0, 0]
  Set speed (120.0 mm/s)
  MoveL (T13422) to (103.84, 109.5, 15.1) mm, rotated rx 180 ry 0 rz -180 deg; joints [0, 0, 0, 0, 0, 0]
  Call Extruder -0.38
  MoveL (T13423) to (103.84, 110.57, 15.1) mm, rotated rx 180 ry 0 rz -180 deg; joints [0, 0, 0, 0, 0, 0]
  Set speed (45.0 mm/s)
  Call Extruder -0.02
  MoveL (T13424) to (103.84, 110.57, 15.1) mm, rotated rx 180 ry 0 rz -180 deg; joints [0, 0, 0, 0, 0, 0]
  Set speed (150.0 mm/s)
  MoveL (T13425) to (103.84, 110.57, 17.1) mm, rotated rx 180 ry 0 rz -180 deg; joints [0, 0, 0, 0, 0, 0]
  MoveL (T13426) to (119.2, 110.57, 17.1) mm, rotated rx 180 ry 0 rz -180 deg; joints [0, 0, 0, 0, 0, 0]
  MoveL (T13427) to (119.2, 110.57, 15.1) mm, rotated rx 180 ry 0 rz -180 deg; joints [0, 0, 0, 0, 0, 0]
  Set speed (40.0 mm/s)
  Call Extruder 2.0
  MoveL (T13428) to (119.2, 110.57, 15.1) mm, rotated rx 180 ry 0 rz -180 deg; joints [0, 0, 0, 0, 0, 0]
  Set speed (28.8 mm/s)
  MoveL (T13429) to (119.2, 110.57, 15.1) mm, rotated rx 180 ry 0 rz -180 deg; joints [0, 0, 0, 0, 0, 0]
  Call Extruder 0.00427
  MoveL (T13430) to (119.1, 110.67, 15.1) mm, rotated rx 180 ry 0 rz -180 deg; joints [0, 0, 0, 0, 0, 0]
  Call Extruder 0.015
  MoveL (T13431) to (119.1, 111.16, 15.1) mm, rotated rx 180 ry 0 rz -180 deg; joints [0, 0, 0, 0, 0, 0]
  Call Extruder 0.01378
  MoveL (T13432) to (119.42, 111.48, 15.1) mm, rotated rx 180 ry 0 rz -180 deg; joints [0, 0, 0, 0, 0, 0]
  Call Extruder 0.03876
  MoveL (T13433) to (120.69, 111.48, 15.1) mm, rotated rx 180 ry 0 rz -180 deg; joints [0, 0, 0, 0, 0, 0]
  Call Extruder 0.02004
  MoveL (T13434) to (121.16, 111.94, 15.1) mm, rotated rx 180 ry 0 rz -180 deg; joints [0, 0, 0, 0, 0, 0]
  Call Extruder 0.01972
  MoveL (T13435) to (121.16, 112.59, 15.1) mm, rotated rx 180 ry 0 rz -180 deg; joints [0, 0, 0, 0, 0, 0]
  Call Extruder 0.05295
  MoveL (T13436) to (119.42, 112.59, 15.1) mm, rotated rx 180 ry 0 rz -180 deg; joints [0, 0, 0, 0, 0, 0]
  Call Extruder 0.00174
  MoveL (T13437) to (119.38, 112.63, 15.1) mm, rotated rx 180 ry 0 rz -180 deg; joints [0, 0, 0, 0, 0, 0]
  Set speed (150.0 mm/s)
  MoveL (T13438) to (120.91, 113.35, 15.1) mm, rotated rx 180 ry 0 rz -180 deg; joints [0, 0, 0, 0, 0, 0]
  Set speed (28.8 mm/s)
  MoveL (T13439) to (120.91, 113.35, 15.1) mm, rotated rx 180 ry 0 rz -180 deg; joints [0, 0, 0, 0, 0, 0]
  Call Extruder 0.01626
  MoveL (T13440) to (120.56, 113, 15.1) mm, rotated rx 180 ry 0 rz -180 deg; joints [0, 0, 0, 0, 0, 0]
  Call Extruder 0.02046
  MoveL (T13441) to (119.94, 113, 15.1) mm, rotated rx 180 ry 0 rz -180 deg; joints [0, 0, 0, 0, 0, 0]
  Call Extruder 0.01626
  MoveL (T13442) to (120.28, 113.35, 15.1) mm, rotated rx 180 ry 0 rz -180 deg; joints [0, 0, 0, 0, 0, 0]
  Set speed (45.0 mm/s)
  Call Extruder -1.6
  MoveL (T13443) to (120.28, 113.35, 15.1) mm, rotated rx 180 ry 0 rz -180 deg; joints [0, 0, 0, 0, 0, 0]
  Set speed (120.0 mm/s)
  MoveL (T13444) to (120.28, 113.35, 15.1) mm, rotated rx 180 ry 0 rz -180 deg; joints [0, 0, 0, 0, 0, 0]
  Call Extruder -0.17616
  MoveL (T13445) to (119.94, 113, 15.1) mm, rotated rx 180 ry 0 rz -180 deg; joints [0, 0, 0, 0, 0, 0]
  Call Extruder -0.20384
  MoveL (T13446) to (120.51, 113, 15.1) mm, rotated rx 180 ry 0 rz -180 deg; joints [0, 0, 0, 0, 0, 0]
  Set speed (45.0 mm/s)
  Call Extruder -0.02
  MoveL (T13447) to (120.51, 113, 15.1) mm, rotated rx 180 ry 0 rz -180 deg; joints [0, 0, 0, 0, 0, 0]
  Set speed (150.0 mm/s)
  MoveL (T13448) to (120.51, 113, 17.1) mm, rotated rx 180 ry 0 rz -180 deg; joints [0, 0, 0, 0, 0, 0]
  MoveL (T13449) to (121.02, 111.25, 17.1) mm, rotated rx 180 ry 0 rz -180 deg; joints [0, 0, 0, 0, 0, 0]
  MoveL (T13450) to (121.02, 111.25, 15.1) mm, rotated rx 180 ry 0 rz -180 deg; joints [0, 0, 0, 0, 0, 0]
  Set speed (40.0 mm/s)
  Call Extruder 2.0
  MoveL (T13451) to (121.02, 111.25, 15.1) mm, rotated rx 180 ry 0 rz -180 deg; joints [0, 0, 0, 0, 0, 0]
  Set speed (28.8 mm/s)
  MoveL (T13452) to (121.02, 111.25, 15.1) mm, rotated rx 180 ry 0 rz -180 deg; joints [0, 0, 0, 0, 0, 0]
  Call Extruder 0.01708
  MoveL (T13453) to (120.64, 110.88, 15.1) mm, rotated rx 180 ry 0 rz -180 deg; joints [0, 0, 0, 0, 0, 0]
  Call Extruder 0.01991
  MoveL (T13454) to (120.03, 110.88, 15.1) mm, rotated rx 180 ry 0 rz -180 deg; joints [0, 0, 0, 0, 0, 0]
  Call Extruder 0.00867
  MoveL (T13455) to (120.22, 111.07, 15.1) mm, rotated rx 180 ry 0 rz -180 deg; joints [0, 0, 0, 0, 0, 0]
  Call Extruder 0.01991
  MoveL (T13456) to (119.61, 111.07, 15.1) mm, rotated rx 180 ry 0 rz -180 deg; joints [0, 0, 0, 0, 0, 0]
  Call Extruder 0.01299
  MoveL (T13457) to (119.32, 110.79, 15.1) mm, rotated rx 180 ry 0 rz -180 deg; joints [0, 0, 0, 0, 0, 0]
  Set speed (45.0 mm/s)
  Call Extruder -1.6
  MoveL (T13458) to (119.32, 110.79, 15.1) mm, rotated rx 180 ry 0 rz -180 deg; joints [0, 0, 0, 0, 0, 0]
  Set speed (120.0 mm/s)
  MoveL (T13459) to (119.32, 110.79, 15.1) mm, rotated rx 180 ry 0 rz -180 deg; joints [0, 0, 0, 0, 0, 0]
  Call Extruder -0.1426
  MoveL (T13460) to (119.61, 111.07, 15.1) mm, rotated rx 180 ry 0 rz -180 deg; joints [0, 0, 0, 0, 0, 0]
  Call Extruder -0.21845
  MoveL (T13461) to (120.22, 111.07, 15.1) mm, rotated rx 180 ry 0 rz -180 deg; joints [0, 0, 0, 0, 0, 0]
  Call Extruder -0.01895
  MoveL (T13462) to (120.18, 111.03, 15.1) mm, rotated rx 180 ry 0 rz -180 deg; joints [0, 0, 0, 0, 0, 0]
  Set speed (45.0 mm/s)
  Call Extruder -0.02
  MoveL (T13463) to (120.18, 111.03, 15.1) mm, rotated rx 180 ry 0 rz -180 deg; joints [0, 0, 0, 0, 0, 0]
  Set speed (150.0 mm/s)
  MoveL (T13464) to (120.18, 111.03, 17.1) mm, rotated rx 180 ry 0 rz -180 deg; joints [0, 0, 0, 0, 0, 0]
  MoveL (T13465) to (120.36, 106.08, 17.1) mm, rotated rx 180 ry 0 rz -180 deg; joints [0, 0, 0, 0, 0, 0]
  MoveL (T13466) to (120.36, 106.08, 15.1) mm, rotated rx 180 ry 0 rz -180 deg; joints [0, 0, 0, 0, 0, 0]
  Set speed (40.0 mm/s)
  Call Extruder 2.0
  MoveL (T13467) to (120.36, 106.08, 15.1) mm, rotated rx 180 ry 0 rz -180 deg; joints [0, 0, 0, 0, 0, 0]
  Set speed (28.8 mm/s)
  MoveL (T13468) to (120.36, 106.08, 15.1) mm, rotated rx 180 ry 0 rz -180 deg; joints [0, 0, 0, 0, 0, 0]
  Call Extruder 0.01802
  MoveL (T13469) to (120.75, 106.47, 15.1) mm, rotated rx 180 ry 0 rz -180 deg; joints [0, 0, 0, 0, 0, 0]
  Call Extruder 0.02094
  MoveL (T13470) to (120.12, 106.47, 15.1) mm, rotated rx 180 ry 0 rz -180 deg; joints [0, 0, 0, 0, 0, 0]
  Call Extruder 0.01802
  MoveL (T13471) to (119.73, 106.08, 15.1) mm, rotated rx 180 ry 0 rz -180 deg; joints [0, 0, 0, 0, 0, 0]
  Set speed (45.0 mm/s)
  Call Extruder -1.6
  MoveL (T13472) to (119.73, 106.08, 15.1) mm, rotated rx 180 ry 0 rz -180 deg; joints [0, 0, 0, 0, 0, 0]
  Set speed (120.0 mm/s)
  MoveL (T13473) to (119.73, 106.08, 15.1) mm, rotated rx 180 ry 0 rz -180 deg; joints [0, 0, 0, 0, 0, 0]
  Call Extruder -0.19276
  MoveL (T13474) to (120.12, 106.47, 15.1) mm, rotated rx 180 ry 0 rz -180 deg; joints [0, 0, 0, 0, 0, 0]
  Call Extruder -0.18724
  MoveL (T13475) to (120.64, 106.47, 15.1) mm, rotated rx 180 ry 0 rz -180 deg; joints [0, 0, 0, 0, 0, 0]
  Set speed (45.0 mm/s)
  Call Extruder -0.02
  MoveL (T13476) to (120.64, 106.47, 15.1) mm, rotated rx 180 ry 0 rz -180 deg; joints [0, 0, 0, 0, 0, 0]
  Set speed (150.0 mm/s)
  MoveL (T13477) to (120.64, 106.47, 17.1) mm, rotated rx 180 ry 0 rz -180 deg; joints [0, 0, 0, 0, 0, 0]
  MoveL (T13478) to (121.08, 118.03, 17.1) mm, rotated rx 180 ry 0 rz -180 deg; joints [0, 0, 0, 0, 0, 0]
  MoveL (T13479) to (121.08, 118.03, 15.1) mm, rotated rx 180 ry 0 rz -180 deg; joints [0, 0, 0, 0, 0, 0]
  Set speed (40.0 mm/s)
  Call Extruder 2.0
  MoveL (T13480) to (121.08, 118.03, 15.1) mm, rotated rx 180 ry 0 rz -180 deg; joints [0, 0, 0, 0, 0, 0]
  Set speed (28.8 mm/s)
  MoveL (T13481) to (121.08, 118.03, 15.1) mm, rotated rx 180 ry 0 rz -180 deg; joints [0, 0, 0, 0, 0, 0]
  Call Extruder 0.0225
  MoveL (T13482) to (120.61, 117.56, 15.1) mm, rotated rx 180 ry 0 rz -180 deg; joints [0, 0, 0, 0, 0, 0]
  Call Extruder 0.02154
  MoveL (T13483) to (119.97, 117.56, 15.1) mm, rotated rx 180 ry 0 rz -180 deg; joints [0, 0, 0, 0, 0, 0]
  Call Extruder 0.01375
  MoveL (T13484) to (120.25, 117.85, 15.1) mm, rotated rx 180 ry 0 rz -180 deg; joints [0, 0, 0, 0, 0, 0]
  Call Extruder 0.02154
  MoveL (T13485) to (119.62, 117.85, 15.1) mm, rotated rx 180 ry 0 rz -180 deg; joints [0, 0, 0, 0, 0, 0]
  Call Extruder 0.01409
  MoveL (T13486) to (119.32, 117.55, 15.1) mm, rotated rx 180 ry 0 rz -180 deg; joints [0, 0, 0, 0, 0, 0]
  Set speed (45.0 mm/s)
  Call Extruder -1.6
  MoveL (T13487) to (119.32, 117.55, 15.1) mm, rotated rx 180 ry 0 rz -180 deg; joints [0, 0, 0, 0, 0, 0]
  Set speed (120.0 mm/s)
  MoveL (T13488) to (119.32, 117.55, 15.1) mm, rotated rx 180 ry 0 rz -180 deg; joints [0, 0, 0, 0, 0, 0]
  Call Extruder -0.14881
  MoveL (T13489) to (119.62, 117.85, 15.1) mm, rotated rx 180 ry 0 rz -180 deg; joints [0, 0, 0, 0, 0, 0]
  Call Extruder -0.22743
  MoveL (T13490) to (120.25, 117.85, 15.1) mm, rotated rx 180 ry 0 rz -180 deg; joints [0, 0, 0, 0, 0, 0]
  Call Extruder -0.00376
  MoveL (T13491) to (120.25, 117.84, 15.1) mm, rotated rx 180 ry 0 rz -180 deg; joints [0, 0, 0, 0, 0, 0]
  Set speed (45.0 mm/s)
  Call Extruder -0.02
  MoveL (T13492) to (120.25, 117.84, 15.1) mm, rotated rx 180 ry 0 rz -180 deg; joints [0, 0, 0, 0, 0, 0]
  Set speed (150.0 mm/s)
  MoveL (T13493) to (120.25, 117.84, 17.1) mm, rotated rx 180 ry 0 rz -180 deg; joints [0, 0, 0, 0, 0, 0]
  MoveL (T13494) to (104.34, 103.54, 17.1) mm, rotated rx 180 ry 0 rz -180 deg; joints [0, 0, 0, 0, 0, 0]
  MoveL (T13495) to (104.34, 103.54, 15.3) mm, rotated rx 180 ry 0 rz -180 deg; joints [0, 0, 0, 0, 0, 0]
  Set speed (40.0 mm/s)
  Call Extruder 2.0
  MoveL (T13496) to (104.34, 103.54, 15.3) mm, rotated rx 180 ry 0 rz -180 deg; joints [0, 0, 0, 0, 0, 0]
  Set speed (27.4 mm/s)
  MoveL (T13497) to (104.34, 103.54, 15.3) mm, rotated rx 180 ry 0 rz -180 deg; joints [0, 0, 0, 0, 0, 0]
  Call Extruder 0.08593
  MoveL (T13498) to (107.16, 103.54, 15.3) mm, rotated rx 180 ry 0 rz -180 deg; joints [0, 0, 0, 0, 0, 0]
  Call Extruder 0.05791
  MoveL (T13499) to (107.16, 105.44, 15.3) mm, rotated rx 180 ry 0 rz -180 deg; joints [0, 0, 0, 0, 0, 0]
  Call Extruder 0.11367
  MoveL (T13500) to (110.89, 105.44, 15.3) mm, rotated rx 180 ry 0 rz -180 deg; joints [0, 0, 0, 0, 0, 0]
  Call Extruder 0.05791
  MoveL (T13501) to (110.89, 103.54, 15.3) mm, rotated rx 180 ry 0 rz -180 deg; joints [0, 0, 0, 0, 0, 0]
  Call Extruder 0.07751
  MoveL (T13502) to (113.44, 103.54, 15.3) mm, rotated rx 180 ry 0 rz -180 deg; joints [0, 0, 0, 0, 0, 0]
  Call Extruder 0.05791
  MoveL (T13503) to (113.44, 105.44, 15.3) mm, rotated rx 180 ry 0 rz -180 deg; joints [0, 0, 0, 0, 0, 0]
  Call Extruder 0.11337
  MoveL (T13504) to (117.16, 105.44, 15.3) mm, rotated rx 180 ry 0 rz -180 deg; joints [0, 0, 0, 0, 0, 0]
  Call Extruder 0.05791
  MoveL (T13505) to (117.16, 103.54, 15.3) mm, rotated rx 180 ry 0 rz -180 deg; joints [0, 0, 0, 0, 0, 0]
  Call Extruder 0.13111
  MoveL (T13506) to (121.46, 103.54, 15.3) mm, rotated rx 180 ry 0 rz -180 deg; joints [0, 0, 0, 0, 0, 0]
  Call Extruder 0.09478
  MoveL (T13507) to (121.46, 106.65, 15.3) mm, rotated rx 180 ry 0 rz -180 deg; joints [0, 0, 0, 0, 0, 0]
  Call Extruder 0.05866
  MoveL (T13508) to (119.53, 106.65, 15.3) mm, rotated rx 180 ry 0 rz -180 deg; joints [0, 0, 0, 0, 0, 0]
  Call Extruder 0.11607
  MoveL (T13509) to (119.53, 110.46, 15.3) mm, rotated rx 180 ry 0 rz -180 deg; joints [0, 0, 0, 0, 0, 0]
  Call Extruder 0.05872
  MoveL (T13510) to (121.46, 110.46, 15.3) mm, rotated rx 180 ry 0 rz -180 deg; joints [0, 0, 0, 0, 0, 0]
  Call Extruder 0.09508
  MoveL (T13511) to (121.46, 113.58, 15.3) mm, rotated rx 180 ry 0 rz -180 deg; joints [0, 0, 0, 0, 0, 0]
  Call Extruder 0.05876
  MoveL (T13512) to (119.53, 113.58, 15.3) mm, rotated rx 180 ry 0 rz -180 deg; joints [0, 0, 0, 0, 0, 0]
  Call Extruder 0.11545
  MoveL (T13513) to (119.53, 117.37, 15.3) mm, rotated rx 180 ry 0 rz -180 deg; joints [0, 0, 0, 0, 0, 0]
  Call Extruder 0.05881
  MoveL (T13514) to (121.46, 117.37, 15.3) mm, rotated rx 180 ry 0 rz -180 deg; joints [0, 0, 0, 0, 0, 0]
  Call Extruder 0.12458
  MoveL (T13515) to (121.46, 121.46, 15.3) mm, rotated rx 180 ry 0 rz -180 deg; joints [0, 0, 0, 0, 0, 0]
  Call Extruder 0.54596
  MoveL (T13516) to (103.54, 121.46, 15.3) mm, rotated rx 180 ry 0 rz -180 deg; joints [0, 0, 0, 0, 0, 0]
  Call Extruder 0.54596
  MoveL (T13517) to (103.54, 103.54, 15.3) mm, rotated rx 180 ry 0 rz -180 deg; joints [0, 0, 0, 0, 0, 0]
  Call Extruder 0.02254
  MoveL (T13518) to (104.28, 103.54, 15.3) mm, rotated rx 180 ry 0 rz -180 deg; joints [-12.046, 47.993, 6.255, -14.732, -55.151, 8.545]
  Set speed (150.0 mm/s)
  MoveL (T13519) to (103.53, 103.13, 15.3) mm, rotated rx 180 ry 0 rz -180 deg; joints [-12.046, 47.993, 6.255, -14.732, -55.151, 8.545]
  Set speed (27.4 mm/s)
  MoveL (T13520) to (103.53, 103.13, 15.3) mm, rotated rx 180 ry 0 rz -180 deg; joints [-12.046, 47.993, 6.255, -14.732, -55.151, 8.545]
  Call Extruder 0.12292
  MoveL (T13521) to (107.57, 103.13, 15.3) mm, rotated rx 180 ry 0 rz -180 deg; joints [-12.046, 47.993, 6.255, -14.732, -55.151, 8.545]
  Call Extruder 0.05791
  MoveL (T13522) to (107.57, 105.03, 15.3) mm, rotated rx 180 ry 0 rz -180 deg; joints [-12.046, 47.993, 6.255, -14.732, -55.151, 8.545]
  Call Extruder 0.08886
  MoveL (T13523) to (110.48, 105.03, 15.3) mm, rotated rx 180 ry 0 rz -180 deg; joints [-12.046, 47.993, 6.255, -14.732, -55.151, 8.545]
  Call Extruder 0.05791
  MoveL (T13524) to (110.48, 103.13, 15.3) mm, rotated rx 180 ry 0 rz -180 deg; joints [-12.046, 47.993, 6.255, -14.732, -55.151, 8.545]
  Call Extruder 0.1023
  MoveL (T13525) to (113.84, 103.13, 15.3) mm, rotated rx 180 ry 0 rz -180 deg; joints [-12.046, 47.993, 6.255, -14.732, -55.151, 8.545]
  Call Extruder 0.05791
  MoveL (T13526) to (113.84, 105.03, 15.3) mm, rotated rx 180 ry 0 rz -180 deg; joints [-12.046, 47.993, 6.255, -14.732, -55.151, 8.545]
  Call Extruder 0.08857
  MoveL (T13527) to (116.75, 105.03, 15.3) mm, rotated rx 180 ry 0 rz -180 deg; joints [-12.046, 47.993, 6.255, -14.732, -55.151, 8.545]
  Call Extruder 0.05791
  MoveL (T13528) to (116.75, 103.13, 15.3) mm, rotated rx 180 ry 0 rz -180 deg; joints [-12.046, 47.993, 6.255, -14.732, -55.151, 8.545]
  Call Extruder 0.15592
  MoveL (T13529) to (121.87, 103.13, 15.3) mm, rotated rx 180 ry 0 rz -180 deg; joints [-12.046, 47.993, 6.255, -14.732, -55.151, 8.545]
  Call Extruder 0.11958
  MoveL (T13530) to (121.87, 107.06, 15.3) mm, rotated rx 180 ry 0 rz -180 deg; joints [-12.046, 47.993, 6.255, -14.732, -55.151, 8.545]
  Call Extruder 0.05867
  MoveL (T13531) to (119.94, 107.06, 15.3) mm, rotated rx 180 ry 0 rz -180 deg; joints [-12.046, 47.993, 6.255, -14.732, -55.151, 8.545]
  Call Extruder 0.09127
  MoveL (T13532) to (119.94, 110.05, 15.3) mm, rotated rx 180 ry 0 rz -180 deg; joints [-12.046, 47.993, 6.255, -14.732, -55.151, 8.545]
  Call Extruder 0.05871
  MoveL (T13533) to (121.87, 110.05, 15.3) mm, rotated rx 180 ry 0 rz -180 deg; joints [-12.046, 47.993, 6.255, -14.732, -55.151, 8.545]
  Call Extruder 0.1199
  MoveL (T13534) to (121.87, 113.99, 15.3) mm, rotated rx 180 ry 0 rz -180 deg; joints [-12.046, 47.993, 6.255, -14.732, -55.151, 8.545]
  Call Extruder 0.05876
  MoveL (T13535) to (119.94, 113.99, 15.3) mm, rotated rx 180 ry 0 rz -180 deg; joints [-12.046, 47.993, 6.255, -14.732, -55.151, 8.545]
  Call Extruder 0.09065
  MoveL (T13536) to (119.94, 116.96, 15.3) mm, rotated rx 180 ry 0 rz -180 deg; joints [-12.046, 47.712, 6.286, -14.777, -54.909, 8.623]
  Call Extruder 0.0588
  MoveL (T13537) to (121.87, 116.97, 15.3) mm, rotated rx 180 ry 0 rz -180 deg; joints [1, 65.387, -26.737, 1.601, -38.661, -1.25]
  Call Extruder 0.14937
  MoveL (T13538) to (121.87, 121.87, 15.3) mm, rotated rx 180 ry 0 rz -180 deg; joints [1, 65.591, -26.771, 1.595, -38.831, -1.243]
  Call Extruder 0.57077
  MoveL (T13539) to (103.13, 121.87, 15.3) mm, rotated rx 180 ry 0 rz -180 deg; joints [1, 65.591, -26.771, 1.595, -38.831, -1.243]
  Call Extruder 0.57077
  MoveL (T13540) to (103.13, 103.13, 15.3) mm, rotated rx 180 ry 0 rz -180 deg; joints [1, 65.591, -26.771, 1.595, -38.831, -1.243]
  Call Extruder 0.01036
  MoveL (T13541) to (103.47, 103.13, 15.3) mm, rotated rx 180 ry 0 rz -180 deg; joints [1, 65.591, -26.771, 1.595, -38.831, -1.243]
  Set speed (150.0 mm/s)
  MoveL (T13542) to (102.72, 102.81, 15.3) mm, rotated rx 180 ry 0 rz -180 deg; joints [1, 65.591, -26.771, 1.595, -38.831, -1.243]
  Set speed (25.0 mm/s)
  MoveL (T13543) to (102.72, 102.81, 15.3) mm, rotated rx 180 ry 0 rz -180 deg; joints [1, 65.591, -26.771, 1.595, -38.831, -1.243]
  Call Extruder 0.00259
  MoveL (T13544) to (102.72, 102.72, 15.3) mm, rotated rx 180 ry 0 rz -180 deg; joints [1, 65.591, -26.771, 1.595, -38.831, -1.243]
  Call Extruder 0.15992
  MoveL (T13545) to (107.97, 102.72, 15.3) mm, rotated rx 180 ry 0 rz -180 deg; joints [1, 65.591, -26.771, 1.595, -38.831, -1.243]
  Call Extruder 0.05791
  MoveL (T13546) to (107.97, 104.63, 15.3) mm, rotated rx 180 ry 0 rz -180 deg; joints [1, 65.591, -26.771, 1.595, -38.831, -1.243]
  Call Extruder 0.06406
  MoveL (T13547) to (110.08, 104.63, 15.3) mm, rotated rx 180 ry 0 rz -180 deg; joints [1, 65.591, -26.771, 1.595, -38.831, -1.243]
  Call Extruder 0.05791
  MoveL (T13548) to (110.08, 102.72, 15.3) mm, rotated rx 180 ry 0 rz -180 deg; joints [1, 65.591, -26.771, 1.595, -38.831, -1.243]
  Call Extruder 0.12709
  MoveL (T13549) to (114.25, 102.72, 15.3) mm, rotated rx 180 ry 0 rz -180 deg; joints [1, 65.591, -26.771, 1.595, -38.831, -1.243]
  Call Extruder 0.05791
  MoveL (T13550) to (114.25, 104.63, 15.3) mm, rotated rx 180 ry 0 rz -180 deg; joints [1, 65.591, -26.771, 1.595, -38.831, -1.243]
  Call Extruder 0.06377
  MoveL (T13551) to (116.34, 104.63, 15.3) mm, rotated rx 180 ry 0 rz -180 deg; joints [1, 65.591, -26.771, 1.595, -38.831, -1.243]
  Call Extruder 0.05791
  MoveL (T13552) to (116.34, 102.72, 15.3) mm, rotated rx 180 ry 0 rz -180 deg; joints [1, 65.591, -26.771, 1.595, -38.831, -1.243]
  Call Extruder 0.18073
  MoveL (T13553) to (122.28, 102.72, 15.3) mm, rotated rx 180 ry 0 rz -180 deg; joints [0.934, 66.058, -27.65, 1.504, -38.418, -1.178]
  Call Extruder 0.14437
  MoveL (T13554) to (122.28, 107.46, 15.3) mm, rotated rx 180 ry 0 rz -180 deg; joints [0.934, 66.058, -27.65, 1.504, -38.418, -1.178]
  Call Extruder 0.05868
  MoveL (T13555) to (120.35, 107.47, 15.3) mm, rotated rx 180 ry 0 rz -180 deg; joints [0.934, 66.058, -27.65, 1.504, -38.418, -1.178]
  Call Extruder 0.06646
  MoveL (T13556) to (120.35, 109.65, 15.3) mm, rotated rx 180 ry 0 rz -180 deg; joints [0.9, 71.688, -38.244, 1.633, -33.455, -1.363]
  Call Extruder 0.05871
  MoveL (T13557) to (122.28, 109.65, 15.3) mm, rotated rx 180 ry 0 rz -180 deg; joints [0.9, 71.688, -38.244, 1.633, -33.455, -1.363]
  Call Extruder 0.14473
  MoveL (T13558) to (122.28, 114.4, 15.3) mm, rotated rx 180 ry 0 rz -180 deg; joints [0.939, 72.198, -39.204, 1.724, -33.006, -1.446]
  Call Extruder 0.05877
  MoveL (T13559) to (120.35, 114.39, 15.3) mm, rotated rx 180 ry 0 rz -180 deg; joints [0.939, 72.198, -39.204, 1.724, -33.006, -1.446]
  Call Extruder 0.06584
  MoveL (T13560) to (120.34, 116.56, 15.3) mm, rotated rx 180 ry 0 rz -180 deg; joints [0.939, 72.198, -39.204, 1.724, -33.006, -1.446]
  Call Extruder 0.0588
  MoveL (T13561) to (122.28, 116.56, 15.3) mm, rotated rx 180 ry 0 rz -180 deg; joints [1.05, 72.602, -39.963, 1.947, -32.653, -1.639]
  Call Extruder 0.17416
  MoveL (T13562) to (122.28, 122.28, 15.3) mm, rotated rx 180 ry 0 rz -180 deg; joints [1.05, 72.602, -39.963, 1.947, -32.653, -1.639]
  Call Extruder 0.59557
  MoveL (T13563) to (102.72, 122.28, 15.3) mm, rotated rx 180 ry 0 rz -180 deg; joints [1.244, 72.805, -40.346, 2.317, -32.48, -1.955]
  Call Extruder 0.59115
  MoveL (T13564) to (102.72, 102.87, 15.3) mm, rotated rx 180 ry 0 rz -180 deg; joints [1.244, 72.805, -40.346, 2.317, -32.48, -1.955]
  Set speed (150.0 mm/s)
  MoveL (T13565) to (102.78, 102.75, 15.3) mm, rotated rx 180 ry 0 rz -180 deg; joints [1.244, 72.805, -40.346, 2.317, -32.48, -1.955]
  Set speed (45.0 mm/s)
  Call Extruder -1.6
  MoveL (T13566) to (102.78, 102.75, 15.3) mm, rotated rx 180 ry 0 rz -180 deg; joints [3.323, 73.074, -40.853, 6.215, -32.374, -5.255]
  Set speed (120.0 mm/s)
  MoveL (T13567) to (102.78, 102.75, 15.3) mm, rotated rx 180 ry 0 rz -180 deg; joints [3.323, 73.074, -40.853, 6.215, -32.374, -5.255]
  Call Extruder -0.05166
  MoveL (T13568) to (102.72, 102.72, 15.3) mm, rotated rx 180 ry 0 rz -180 deg; joints [3.49, 72.973, -40.661, 6.508, -32.479, -5.497]
  Call Extruder -0.32834
  MoveL (T13569) to (103.65, 102.72, 15.3) mm, rotated rx 180 ry 0 rz -180 deg; joints [3.622, 72.633, -40.022, 6.699, -32.79, -5.639]
  Set speed (45.0 mm/s)
  Call Extruder -0.02
  MoveL (T13570) to (103.65, 102.72, 15.3) mm, rotated rx 180 ry 0 rz -180 deg; joints [3.622, 72.633, -40.022, 6.699, -32.79, -5.639]
  Set speed (150.0 mm/s)
  MoveL (T13571) to (103.65, 102.72, 17.3) mm, rotated rx 180 ry 0 rz -180 deg; joints [3.694, 72.032, -38.891, 6.735, -33.323, -5.636]
  MoveL (T13572) to (106.29, 103.84, 17.3) mm, rotated rx 180 ry 0 rz -180 deg; joints [3.694, 72.032, -38.891, 6.735, -33.323, -5.636]
  MoveL (T13573) to (106.29, 103.84, 15.3) mm, rotated rx 180 ry 0 rz -180 deg; joints [3.694, 72.032, -38.891, 6.735, -33.323, -5.636]
  Set speed (40.0 mm/s)
  Call Extruder 2.0
  MoveL (T13574) to (106.29, 103.84, 15.3) mm, rotated rx 180 ry 0 rz -180 deg; joints [3.834, 66.341, -28.181, 6.19, -38.322, -4.864]
  Set speed (27.4 mm/s)
  MoveL (T13575) to (106.29, 103.84, 15.3) mm, rotated rx 180 ry 0 rz -180 deg; joints [3.834, 66.341, -28.181, 6.19, -38.322, -4.864]
  Call Extruder 0.07441
  MoveL (T13576) to (103.84, 103.84, 15.3) mm, rotated rx 180 ry 0 rz -180 deg; joints [3.834, 66.341, -28.181, 6.19, -38.322, -4.864]
  Call Extruder 0.7458
  MoveL (T13577) to (121.16, 121.16, 15.3) mm, rotated rx 180 ry 0 rz -180 deg; joints [3.803, 65.935, -27.418, 6.092, -38.675, -4.763]
  Call Extruder 0.08828
  MoveL (T13578) to (121.16, 118.26, 15.3) mm, rotated rx 180 ry 0 rz -180 deg; joints [3.803, 65.935, -27.418, 6.092, -38.675, -4.763]
  Call Extruder 0.01815
  MoveL (T13579) to (120.56, 118.26, 15.3) mm, rotated rx 180 ry 0 rz -180 deg; joints [3.693, 65.615, -26.817, 5.881, -38.946, -4.58]
  Call Extruder 0.12488
  MoveL (T13580) to (117.66, 121.16, 15.3) mm, rotated rx 180 ry 0 rz -180 deg; joints [3.693, 65.615, -26.817, 5.881, -38.946, -4.58]
  Call Extruder 0.03385
  MoveL (T13581) to (116.55, 121.16, 15.3) mm, rotated rx 180 ry 0 rz -180 deg; joints [3.493, 65.445, -26.496, 5.545, -39.08, -4.31]
  Call Extruder 0.54738
  MoveL (T13582) to (103.84, 108.45, 15.3) mm, rotated rx 180 ry 0 rz -180 deg; joints [3.493, 65.445, -26.496, 5.545, -39.08, -4.31]
  Call Extruder 0.03385
  MoveL (T13583) to (103.84, 107.34, 15.3) mm, rotated rx 180 ry 0 rz -180 deg; joints [3.493, 65.445, -26.496, 5.545, -39.08, -4.31]
  Call Extruder 0.12966
  MoveL (T13584) to (106.85, 104.33, 15.3) mm, rotated rx 180 ry 0 rz -180 deg; joints [1.308, 65.238, -26.107, 2.071, -39.149, -1.607]
  Call Extruder 0.04315
  MoveL (T13585) to (106.85, 105.75, 15.3) mm, rotated rx 180 ry 0 rz -180 deg; joints [1.308, 65.238, -26.107, 2.071, -39.149, -1.607]
  Call Extruder 0.03126
  MoveL (T13586) to (107.88, 105.75, 15.3) mm, rotated rx 180 ry 0 rz -180 deg; joints [1.134, 65.327, -26.274, 1.8, -39.066, -1.398]
  Set speed (45.0 mm/s)
  Call Extruder -1.6
  MoveL (T13587) to (107.88, 105.75, 15.3) mm, rotated rx 180 ry 0 rz -180 deg; joints [1.134, 65.327, -26.274, 1.8, -39.066, -1.398]
  Set speed (120.0 mm/s)
  MoveL (T13588) to (107.88, 105.75, 15.3) mm, rotated rx 180 ry 0 rz -180 deg; joints [1.005, 65.581, -26.753, 1.603, -38.839, -1.249]
  Call Extruder -0.36558
  MoveL (T13589) to (106.85, 105.75, 15.3) mm, rotated rx 180 ry 0 rz -180 deg; joints [1.005, 65.581, -26.753, 1.603, -38.839, -1.249]
  Call Extruder -0.01442
  MoveL (T13590) to (106.85, 105.7, 15.3) mm, rotated rx 180 ry 0 rz -180 deg; joints [1.005, 65.581, -26.753, 1.603, -38.839, -1.249]
  Set speed (45.0 mm/s)
  Call Extruder -0.02
  MoveL (T13591) to (106.85, 105.7, 15.3) mm, rotated rx 180 ry 0 rz -180 deg; joints [1.005, 65.581, -26.753, 1.603, -38.839, -1.249]
  Set speed (150.0 mm/s)
  MoveL (T13592) to (106.85, 105.7, 17.3) mm, rotated rx 180 ry 0 rz -180 deg; joints [1.005, 65.581, -26.753, 1.603, -38.839, -1.249]
  MoveL (T13593) to (111.01, 105.87, 17.3) mm, rotated rx 180 ry 0 rz -180 deg; joints [1.005, 65.581, -26.753, 1.603, -38.839, -1.249]
  MoveL (T13594) to (111.01, 105.87, 15.3) mm, rotated rx 180 ry 0 rz -180 deg; joints [1.005, 65.581, -26.753, 1.603, -38.839, -1.249]
  Set speed (40.0 mm/s)
  Call Extruder 2.0
  MoveL (T13595) to (111.01, 105.87, 15.3) mm, rotated rx 180 ry 0 rz -180 deg; joints [1.005, 65.581, -26.753, 1.603, -38.839, -1.249]
  Set speed (27.4 mm/s)
  MoveL (T13596) to (111.01, 105.87, 15.3) mm, rotated rx 180 ry 0 rz -180 deg; joints [1.005, 65.581, -26.753, 1.603, -38.839, -1.249]
  Call Extruder 0.01372
  MoveL (T13597) to (111.46, 105.87, 15.3) mm, rotated rx 180 ry 0 rz -180 deg; joints [1.005, 65.581, -26.753, 1.603, -38.839, -1.249]
  Call Extruder 0.01375
  MoveL (T13598) to (111.78, 105.55, 15.3) mm, rotated rx 180 ry 0 rz -180 deg; joints [0.968, 65.833, -27.227, 1.55, -38.616, -1.211]
  Call Extruder 0.04694
  MoveL (T13599) to (111.78, 104.01, 15.3) mm, rotated rx 180 ry 0 rz -180 deg; joints [0.968, 65.833, -27.227, 1.55, -38.616, -1.211]
  Call Extruder 0.00724
  MoveL (T13600) to (111.94, 103.84, 15.3) mm, rotated rx 180 ry 0 rz -180 deg; joints [0.968, 65.833, -27.227, 1.55, -38.616, -1.211]
  Call Extruder 0.01684
  MoveL (T13601) to (112.5, 103.84, 15.3) mm, rotated rx 180 ry 0 rz -180 deg; joints [0.968, 65.833, -27.227, 1.55, -38.616, -1.211]
  Call Extruder 0.05207
  MoveL (T13602) to (112.5, 105.55, 15.3) mm, rotated rx 180 ry 0 rz -180 deg; joints [0.968, 65.594, -27.187, 1.557, -38.417, -1.22]
  Call Extruder 0.0055
  MoveL (T13603) to (112.63, 105.68, 15.3) mm, rotated rx 180 ry 0 rz -180 deg; joints [1.332, 65.916, -27.792, 2.157, -38.144, -1.697]
  Set speed (150.0 mm/s)
  MoveL (T13604) to (113.31, 104.67, 15.3) mm, rotated rx 180 ry 0 rz -180 deg; joints [1.332, 66.155, -27.832, 2.148, -38.343, -1.685]
  Set speed (27.4 mm/s)
  MoveL (T13605) to (113.31, 104.67, 15.3) mm, rotated rx 180 ry 0 rz -180 deg; joints [1.332, 66.155, -27.832, 2.148, -38.343, -1.685]
  Call Extruder 0.01928
  MoveL (T13606) to (112.91, 105.08, 15.3) mm, rotated rx 180 ry 0 rz -180 deg; joints [1.332, 66.155, -27.832, 2.148, -38.343, -1.685]
  Call Extruder 0.02097
  MoveL (T13607) to (112.9, 104.45, 15.3) mm, rotated rx 180 ry 0 rz -180 deg; joints [1.332, 66.155, -27.832, 2.148, -38.343, -1.685]
  Call Extruder 0.01928
  MoveL (T13608) to (113.31, 104.04, 15.3) mm, rotated rx 180 ry 0 rz -180 deg; joints [1.332, 66.155, -27.832, 2.148, -38.343, -1.685]
  Set speed (45.0 mm/s)
  Call Extruder -1.6
  MoveL (T13609) to (113.31, 104.04, 15.3) mm, rotated rx 180 ry 0 rz -180 deg; joints [1.332, 66.155, -27.832, 2.148, -38.343, -1.685]
  Set speed (120.0 mm/s)
  MoveL (T13610) to (113.31, 104.04, 15.3) mm, rotated rx 180 ry 0 rz -180 deg; joints [1.332, 66.155, -27.832, 2.148, -38.343, -1.685]
  Call Extruder -0.20613
  MoveL (T13611) to (112.9, 104.45, 15.3) mm, rotated rx 180 ry 0 rz -180 deg; joints [1.332, 66.155, -27.832, 2.148, -38.343, -1.685]
  Call Extruder -0.17387
  MoveL (T13612) to (112.91, 104.94, 15.3) mm, rotated rx 180 ry 0 rz -180 deg; joints [1.332, 66.155, -27.832, 2.148, -38.343, -1.685]
  Set speed (45.0 mm/s)
  Call Extruder -0.02
  MoveL (T13613) to (112.91, 104.94, 15.3) mm, rotated rx 180 ry 0 rz -180 deg; joints [1.332, 66.155, -27.832, 2.148, -38.343, -1.685]
  Set speed (150.0 mm/s)
  MoveL (T13614) to (112.91, 104.94, 17.3) mm, rotated rx 180 ry 0 rz -180 deg; joints [1.332, 66.155, -27.832, 2.148, -38.343, -1.685]
  MoveL (T13615) to (111.09, 105.65, 17.3) mm, rotated rx 180 ry 0 rz -180 deg; joints [1.285, 71.612, -38.101, 2.327, -33.533, -1.94]
  MoveL (T13616) to (111.09, 105.65, 15.3) mm, rotated rx 180 ry 0 rz -180 deg; joints [1.285, 71.612, -38.101, 2.327, -33.533, -1.94]
  Set speed (40.0 mm/s)
  Call Extruder 2.0
  MoveL (T13617) to (111.09, 105.65, 15.3) mm, rotated rx 180 ry 0 rz -180 deg; joints [1.285, 71.612, -38.101, 2.327, -33.533, -1.94]
  Set speed (27.4 mm/s)
  MoveL (T13618) to (111.09, 105.65, 15.3) mm, rotated rx 180 ry 0 rz -180 deg; joints [3.313, 71.86, -38.568, 6.02, -33.438, -5.03]
  Call Extruder 0.0125
  MoveL (T13619) to (111.37, 105.37, 15.3) mm, rotated rx 180 ry 0 rz -180 deg; joints [3.313, 71.86, -38.568, 6.02, -33.438, -5.03]
  Call Extruder 0.01918
  MoveL (T13620) to (111.37, 104.77, 15.3) mm, rotated rx 180 ry 0 rz -180 deg; joints [3.435, 66.36, -28.218, 5.551, -38.273, -4.363]
  Call Extruder 0.0078
  MoveL (T13621) to (111.2, 104.94, 15.3) mm, rotated rx 180 ry 0 rz -180 deg; joints [3.435, 66.36, -28.218, 5.551, -38.273, -4.363]
  Call Extruder 0.01918
  MoveL (T13622) to (111.2, 104.34, 15.3) mm, rotated rx 180 ry 0 rz -180 deg; joints [1.339, 66.155, -27.833, 2.158, -38.342, -1.693]
  Call Extruder 0.01606
  MoveL (T13623) to (111.55, 103.98, 15.3) mm, rotated rx 180 ry 0 rz -180 deg; joints [1.339, 66.155, -27.833, 2.158, -38.342, -1.693]
  Set speed (45.0 mm/s)
  Call Extruder -1.6
  MoveL (T13624) to (111.55, 103.98, 15.3) mm, rotated rx 180 ry 0 rz -180 deg; joints [1.343, 66.254, -28.018, 2.169, -38.256, -1.703]
  Set speed (120.0 mm/s)
  MoveL (T13625) to (111.55, 103.98, 15.3) mm, rotated rx 180 ry 0 rz -180 deg; joints [1.343, 66.254, -28.018, 2.169, -38.256, -1.703]
  Call Extruder -0.17962
  MoveL (T13626) to (111.2, 104.34, 15.3) mm, rotated rx 180 ry 0 rz -180 deg; joints [1.343, 66.254, -28.018, 2.169, -38.256, -1.703]
  Call Extruder -0.20038
  MoveL (T13627) to (111.2, 104.9, 15.3) mm, rotated rx 180 ry 0 rz -180 deg; joints [1.343, 66.254, -28.018, 2.169, -38.256, -1.703]
  Set speed (45.0 mm/s)
  Call Extruder -0.02
  MoveL (T13628) to (111.2, 104.9, 15.3) mm, rotated rx 180 ry 0 rz -180 deg; joints [1.343, 66.254, -28.018, 2.169, -38.256, -1.703]
  Set speed (150.0 mm/s)
  MoveL (T13629) to (111.2, 104.9, 17.3) mm, rotated rx 180 ry 0 rz -180 deg; joints [1.343, 66.254, -28.018, 2.169, -38.256, -1.703]
  MoveL (T13630) to (117.12, 105.75, 17.3) mm, rotated rx 180 ry 0 rz -180 deg; joints [1.343, 66.254, -28.018, 2.169, -38.256, -1.703]
  MoveL (T13631) to (117.12, 105.75, 15.3) mm, rotated rx 180 ry 0 rz -180 deg; joints [1.343, 66.254, -28.018, 2.169, -38.256, -1.703]
  Set speed (40.0 mm/s)
  Call Extruder 2.0
  MoveL (T13632) to (117.12, 105.75, 15.3) mm, rotated rx 180 ry 0 rz -180 deg; joints [1.336, 66.427, -28.344, 2.165, -38.103, -1.704]
  Set speed (27.4 mm/s)
  MoveL (T13633) to (117.12, 105.75, 15.3) mm, rotated rx 180 ry 0 rz -180 deg; joints [1.336, 66.427, -28.344, 2.165, -38.103, -1.704]
  Call Extruder 0.01044
  MoveL (T13634) to (117.46, 105.75, 15.3) mm, rotated rx 180 ry 0 rz -180 deg; joints [1.336, 66.427, -28.344, 2.165, -38.103, -1.704]
  Call Extruder 0.05791
  MoveL (T13635) to (117.46, 103.84, 15.3) mm, rotated rx 180 ry 0 rz -180 deg; joints [1.336, 66.427, -28.344, 2.165, -38.103, -1.704]
  Call Extruder 0.00606
  MoveL (T13636) to (117.66, 103.84, 15.3) mm, rotated rx 180 ry 0 rz -180 deg; joints [1.336, 66.427, -28.344, 2.165, -38.103, -1.704]
  Call Extruder 0.10776
  MoveL (T13637) to (120.16, 106.35, 15.3) mm, rotated rx 180 ry 0 rz -180 deg; joints [1.336, 66.189, -28.304, 2.174, -37.905, -1.716]
  Call Extruder 0.03025
  MoveL (T13638) to (121.16, 106.34, 15.3) mm, rotated rx 180 ry 0 rz -180 deg; joints [3.278, 71.505, -38.293, 5.97, -33.355, -4.992]
  Call Extruder 0.07618
  MoveL (T13639) to (121.16, 103.84, 15.3) mm, rotated rx 180 ry 0 rz -180 deg; joints [3.278, 71.74, -38.341, 5.94, -33.541, -4.957]
  Call Extruder 0.7458
  MoveL (T13640) to (103.84, 121.16, 15.3) mm, rotated rx 180 ry 0 rz -180 deg; joints [3.278, 71.74, -38.341, 5.94, -33.541, -4.957]
  Call Extruder 0.10645
  MoveL (T13641) to (103.84, 117.66, 15.3) mm, rotated rx 180 ry 0 rz -180 deg; joints [3.278, 71.74, -38.341, 5.94, -33.541, -4.957]
  Call Extruder 0.15054
  MoveL (T13642) to (107.34, 121.16, 15.3) mm, rotated rx 180 ry 0 rz -180 deg; joints [3.278, 71.74, -38.341, 5.94, -33.541, -4.957]
  Call Extruder 0.03385
  MoveL (T13643) to (108.45, 121.16, 15.3) mm, rotated rx 180 ry 0 rz -180 deg; joints [3.278, 71.74, -38.341, 5.94, -33.541, -4.957]
  Call Extruder 0.46435
  MoveL (T13644) to (119.23, 110.38, 15.3) mm, rotated rx 180 ry 0 rz -180 deg; joints [3.278, 71.74, -38.341, 5.94, -33.541, -4.957]
  Call Extruder 0.01097
  MoveL (T13645) to (119.23, 110.02, 15.3) mm, rotated rx 180 ry 0 rz -180 deg; joints [3.278, 71.74, -38.341, 5.94, -33.541, -4.957]
  Call Extruder 0.18404
  MoveL (T13646) to (114.96, 105.75, 15.3) mm, rotated rx 180 ry 0 rz -180 deg; joints [3.278, 71.74, -38.341, 5.94, -33.541, -4.957]
  Call Extruder 0.00937
  MoveL (T13647) to (114.65, 105.75, 15.3) mm, rotated rx 180 ry 0 rz -180 deg; joints [3.278, 71.74, -38.341, 5.94, -33.541, -4.957]
  Call Extruder 0.46549
  MoveL (T13648) to (103.84, 116.55, 15.3) mm, rotated rx 180 ry 0 rz -180 deg; joints [3.278, 71.74, -38.341, 5.94, -33.541, -4.957]
  Call Extruder 0.10645
  MoveL (T13649) to (103.84, 113.06, 15.3) mm, rotated rx 180 ry 0 rz -180 deg; joints [3.278, 71.74, -38.341, 5.94, -33.541, -4.957]
  Call Extruder 0.34896
  MoveL (T13650) to (111.94, 121.16, 15.3) mm, rotated rx 180 ry 0 rz -180 deg; joints [3.394, 66.446, -28.379, 5.494, -38.195, -4.323]
  Call Extruder 0.03385
  MoveL (T13651) to (113.06, 121.16, 15.3) mm, rotated rx 180 ry 0 rz -180 deg; joints [3.394, 66.446, -28.379, 5.494, -38.195, -4.323]
  Call Extruder 0.26584
  MoveL (T13652) to (119.23, 114.98, 15.3) mm, rotated rx 180 ry 0 rz -180 deg; joints [1.37, 66.248, -28.006, 2.213, -38.262, -1.738]
  Call Extruder 0.0111
  MoveL (T13653) to (119.23, 114.62, 15.3) mm, rotated rx 180 ry 0 rz -180 deg; joints [1.37, 66.248, -28.006, 2.213, -38.262, -1.738]
  Call Extruder 0.38237
  MoveL (T13654) to (110.35, 105.75, 15.3) mm, rotated rx 180 ry 0 rz -180 deg; joints [1.37, 66.248, -28.006, 2.213, -38.262, -1.738]
  Call Extruder 0.00937
  MoveL (T13655) to (110.04, 105.75, 15.3) mm, rotated rx 180 ry 0 rz -180 deg; joints [1.323, 71.502, -37.894, 2.389, -33.631, -1.99]
  Call Extruder 0.26707
  MoveL (T13656) to (103.84, 111.94, 15.3) mm, rotated rx 180 ry 0 rz -180 deg; joints [1.323, 71.502, -37.894, 2.389, -33.631, -1.99]
  Call Extruder 0.07441
  MoveL (T13657) to (103.84, 109.5, 15.3) mm, rotated rx 180 ry 0 rz -180 deg; joints [1.323, 71.502, -37.894, 2.389, -33.631, -1.99]
  Set speed (45.0 mm/s)
  Call Extruder -1.6
  MoveL (T13658) to (103.84, 109.5, 15.3) mm, rotated rx 180 ry 0 rz -180 deg; joints [3.272, 71.739, -38.339, 5.929, -33.541, -4.947]
  Set speed (120.0 mm/s)
  MoveL (T13659) to (103.84, 109.5, 15.3) mm, rotated rx 180 ry 0 rz -180 deg; joints [3.243, 71.621, -38.117, 5.861, -33.642, -4.885]
  Call Extruder -0.38
  MoveL (T13660) to (103.84, 110.57, 15.3) mm, rotated rx 180 ry 0 rz -180 deg; joints [3.243, 71.621, -38.117, 5.861, -33.642, -4.885]
  Set speed (45.0 mm/s)
  Call Extruder -0.02
  MoveL (T13661) to (103.84, 110.57, 15.3) mm, rotated rx 180 ry 0 rz -180 deg; joints [3.243, 71.621, -38.117, 5.861, -33.642, -4.885]
  Set speed (150.0 mm/s)
  MoveL (T13662) to (103.84, 110.57, 17.3) mm, rotated rx 180 ry 0 rz -180 deg; joints [3.243, 71.621, -38.117, 5.861, -33.642, -4.885]
  MoveL (T13663) to (119.11, 110.53, 17.3) mm, rotated rx 180 ry 0 rz -180 deg; joints [3.243, 71.621, -38.117, 5.861, -33.642, -4.885]
  MoveL (T13664) to (119.11, 110.53, 15.3) mm, rotated rx 180 ry 0 rz -180 deg; joints [3.353, 66.532, -28.54, 5.437, -38.117, -4.283]
  Set speed (40.0 mm/s)
  Call Extruder 2.0
  MoveL (T13665) to (119.11, 110.53, 15.3) mm, rotated rx 180 ry 0 rz -180 deg; joints [3.353, 66.532, -28.54, 5.437, -38.117, -4.283]
  Set speed (27.4 mm/s)
  MoveL (T13666) to (119.11, 110.53, 15.3) mm, rotated rx 180 ry 0 rz -180 deg; joints [3.353, 66.532, -28.54, 5.437, -38.117, -4.283]
  Call Extruder 0.00071
  MoveL (T13667) to (119.1, 110.55, 15.3) mm, rotated rx 180 ry 0 rz -180 deg; joints [1.408, 66.34, -28.181, 2.277, -38.182, -1.79]
  Call Extruder 0.015
  MoveL (T13668) to (119.1, 111.04, 15.3) mm, rotated rx 180 ry 0 rz -180 deg; joints [1.408, 66.34, -28.181, 2.277, -38.182, -1.79]
  Call Extruder 0.01378
  MoveL (T13669) to (119.42, 111.36, 15.3) mm, rotated rx 180 ry 0 rz -180 deg; joints [1.408, 66.34, -28.181, 2.277, -38.182, -1.79]
  Call Extruder 0.03519
  MoveL (T13670) to (120.57, 111.36, 15.3) mm, rotated rx 180 ry 0 rz -180 deg; joints [1.361, 71.393, -37.689, 2.452, -33.729, -2.04]
  Call Extruder 0.02508
  MoveL (T13671) to (121.16, 111.94, 15.3) mm, rotated rx 180 ry 0 rz -180 deg; joints [1.361, 71.393, -37.689, 2.452, -33.729, -2.04]
  Call Extruder 0.0231
  MoveL (T13672) to (121.16, 112.7, 15.3) mm, rotated rx 180 ry 0 rz -180 deg; joints [1.361, 71.393, -37.689, 2.452, -33.729, -2.04]
  Call Extruder 0.0513
  MoveL (T13673) to (119.47, 112.7, 15.3) mm, rotated rx 180 ry 0 rz -180 deg; joints [3.237, 71.62, -38.115, 5.85, -33.643, -4.875]
  Set speed (150.0 mm/s)
  MoveL (T13674) to (121, 112.93, 15.3) mm, rotated rx 180 ry 0 rz -180 deg; joints [3.237, 71.62, -38.115, 5.85, -33.643, -4.875]
  Set speed (27.4 mm/s)
  MoveL (T13675) to (121, 112.93, 15.3) mm, rotated rx 180 ry 0 rz -180 deg; joints [3.237, 71.62, -38.115, 5.85, -33.643, -4.875]
  Call Extruder 0.01588
  MoveL (T13676) to (120.65, 113.28, 15.3) mm, rotated rx 180 ry 0 rz -180 deg; joints [3.237, 71.62, -38.115, 5.85, -33.643, -4.875]
  Call Extruder 0.01956
  MoveL (T13677) to (120.04, 113.27, 15.3) mm, rotated rx 180 ry 0 rz -180 deg; joints [3.237, 71.62, -38.115, 5.85, -33.643, -4.875]
  Call Extruder 0.00755
  MoveL (T13678) to (120.21, 113.11, 15.3) mm, rotated rx 180 ry 0 rz -180 deg; joints [3.237, 71.62, -38.115, 5.85, -33.643, -4.875]
  Call Extruder 0.01956
  MoveL (T13679) to (119.6, 113.11, 15.3) mm, rotated rx 180 ry 0 rz -180 deg; joints [3.237, 71.62, -38.115, 5.85, -33.643, -4.875]
  Call Extruder 0.01277
  MoveL (T13680) to (119.32, 113.39, 15.3) mm, rotated rx 180 ry 0 rz -180 deg; joints [3.237, 71.62, -38.115, 5.85, -33.643, -4.875]
  Set speed (45.0 mm/s)
  Call Extruder -1.6
  MoveL (T13681) to (119.32, 113.39, 15.3) mm, rotated rx 180 ry 0 rz -180 deg; joints [3.244, 71.285, -37.484, 5.817, -33.937, -4.831]
  Set speed (120.0 mm/s)
  MoveL (T13682) to (119.32, 113.39, 15.3) mm, rotated rx 180 ry 0 rz -180 deg; joints [3.244, 71.285, -37.484, 5.817, -33.937, -4.831]
  Call Extruder -0.1413
  MoveL (T13683) to (119.6, 113.11, 15.3) mm, rotated rx 180 ry 0 rz -180 deg; joints [3.244, 71.285, -37.484, 5.817, -33.937, -4.831]
  Call Extruder -0.21643
  MoveL (T13684) to (120.21, 113.11, 15.3) mm, rotated rx 180 ry 0 rz -180 deg; joints [3.244, 71.285, -37.484, 5.817, -33.937, -4.831]
  Call Extruder -0.02227
  MoveL (T13685) to (120.17, 113.15, 15.3) mm, rotated rx 180 ry 0 rz -180 deg; joints [3.244, 71.285, -37.484, 5.817, -33.937, -4.831]
  Set speed (45.0 mm/s)
  Call Extruder -0.02
  MoveL (T13686) to (120.17, 113.15, 15.3) mm, rotated rx 180 ry 0 rz -180 deg; joints [3.244, 71.285, -37.484, 5.817, -33.937, -4.831]
  Set speed (150.0 mm/s)
  MoveL (T13687) to (120.17, 113.15, 17.3) mm, rotated rx 180 ry 0 rz -180 deg; joints [3.244, 71.049, -37.437, 5.845, -33.75, -4.865]
  MoveL (T13688) to (120.92, 110.58, 17.3) mm, rotated rx 180 ry 0 rz -180 deg; joints [1.375, 71.134, -37.201, 2.461, -33.957, -2.042]
  MoveL (T13689) to (120.92, 110.58, 15.3) mm, rotated rx 180 ry 0 rz -180 deg; joints [1.375, 71.134, -37.201, 2.461, -33.957, -2.042]
  Set speed (40.0 mm/s)
  Call Extruder 2.0
  MoveL (T13690) to (120.92, 110.58, 15.3) mm, rotated rx 180 ry 0 rz -180 deg; joints [1.375, 71.134, -37.201, 2.461, -33.957, -2.042]
  Set speed (27.4 mm/s)
  MoveL (T13691) to (120.92, 110.58, 15.3) mm, rotated rx 180 ry 0 rz -180 deg; joints [1.375, 71.134, -37.201, 2.461, -33.957, -2.042]
  Call Extruder 0.01747
  MoveL (T13692) to (120.55, 110.95, 15.3) mm, rotated rx 180 ry 0 rz -180 deg; joints [1.375, 71.134, -37.201, 2.461, -33.957, -2.042]
  Call Extruder 0.02082
  MoveL (T13693) to (119.92, 110.95, 15.3) mm, rotated rx 180 ry 0 rz -180 deg; joints [1.375, 71.134, -37.201, 2.461, -33.957, -2.042]
  Call Extruder 0.01747
  MoveL (T13694) to (120.3, 110.58, 15.3) mm, rotated rx 180 ry 0 rz -180 deg; joints [1.375, 71.134, -37.201, 2.461, -33.957, -2.042]
  Set speed (45.0 mm/s)
  Call Extruder -1.6
  MoveL (T13695) to (120.3, 110.58, 15.3) mm, rotated rx 180 ry 0 rz -180 deg; joints [1.375, 71.134, -37.201, 2.461, -33.957, -2.042]
  Set speed (120.0 mm/s)
  MoveL (T13696) to (120.3, 110.58, 15.3) mm, rotated rx 180 ry 0 rz -180 deg; joints [1.375, 71.134, -37.201, 2.461, -33.957, -2.042]
  Call Extruder -0.18758
  MoveL (T13697) to (119.92, 110.95, 15.3) mm, rotated rx 180 ry 0 rz -180 deg; joints [1.375, 71.134, -37.201, 2.461, -33.957, -2.042]
  Call Extruder -0.19242
  MoveL (T13698) to (120.46, 110.95, 15.3) mm, rotated rx 180 ry 0 rz -180 deg; joints [1.375, 71.134, -37.201, 2.461, -33.957, -2.042]
  Set speed (45.0 mm/s)
  Call Extruder -0.02
  MoveL (T13699) to (120.46, 110.95, 15.3) mm, rotated rx 180 ry 0 rz -180 deg; joints [1.433, 71.315, -37.541, 2.576, -33.8, -2.141]
  Set speed (150.0 mm/s)
  MoveL (T13700) to (120.46, 110.95, 17.3) mm, rotated rx 180 ry 0 rz -180 deg; joints [1.486, 71.319, -37.549, 2.672, -33.799, -2.221]
  MoveL (T13701) to (120.91, 117.49, 17.3) mm, rotated rx 180 ry 0 rz -180 deg; joints [1.486, 71.319, -37.549, 2.672, -33.799, -2.221]
  MoveL (T13702) to (120.91, 117.49, 15.3) mm, rotated rx 180 ry 0 rz -180 deg; joints [1.486, 71.319, -37.549, 2.672, -33.799, -2.221]
  Set speed (40.0 mm/s)
  Call Extruder 2.0
  MoveL (T13703) to (120.91, 117.49, 15.3) mm, rotated rx 180 ry 0 rz -180 deg; joints [1.392, 71.028, -37.001, 2.487, -34.052, -2.061]
  Set speed (27.4 mm/s)
  MoveL (T13704) to (120.91, 117.49, 15.3) mm, rotated rx 180 ry 0 rz -180 deg; joints [1.392, 71.028, -37.001, 2.487, -34.052, -2.061]
  Call Extruder 0.01669
  MoveL (T13705) to (120.56, 117.85, 15.3) mm, rotated rx 180 ry 0 rz -180 deg; joints [1.392, 71.028, -37.001, 2.487, -34.052, -2.061]
  Call Extruder 0.0206
  MoveL (T13706) to (119.93, 117.85, 15.3) mm, rotated rx 180 ry 0 rz -180 deg; joints [1.394, 70.872, -36.707, 2.48, -34.189, -2.052]
  Call Extruder 0.01669
  MoveL (T13707) to (120.29, 117.49, 15.3) mm, rotated rx 180 ry 0 rz -180 deg; joints [1.394, 70.872, -36.707, 2.48, -34.189, -2.052]
  Set speed (45.0 mm/s)
  Call Extruder -1.6
  MoveL (T13708) to (120.29, 117.49, 15.3) mm, rotated rx 180 ry 0 rz -180 deg; joints [1.539, 71.323, -37.557, 2.768, -33.797, -2.301]
  Set speed (120.0 mm/s)
  MoveL (T13709) to (120.29, 117.49, 15.3) mm, rotated rx 180 ry 0 rz -180 deg; joints [1.539, 71.323, -37.557, 2.768, -33.797, -2.301]
  Call Extruder -0.17994
  MoveL (T13710) to (119.93, 117.85, 15.3) mm, rotated rx 180 ry 0 rz -180 deg; joints [1.539, 71.323, -37.557, 2.768, -33.797, -2.301]
  Call Extruder -0.20006
  MoveL (T13711) to (120.49, 117.85, 15.3) mm, rotated rx 180 ry 0 rz -180 deg; joints [1.539, 71.323, -37.557, 2.768, -33.797, -2.301]
  Set speed (45.0 mm/s)
  Call Extruder -0.02
  MoveL (T13712) to (120.49, 117.85, 15.3) mm, rotated rx 180 ry 0 rz -180 deg; joints [1.592, 71.327, -37.565, 2.864, -33.796, -2.381]
  Set speed (150.0 mm/s)
  MoveL (T13713) to (120.49, 117.85, 17.3) mm, rotated rx 180 ry 0 rz -180 deg; joints [1.592, 71.327, -37.565, 2.864, -33.796, -2.381]
  MoveL (T13714) to (104.34, 103.54, 17.3) mm, rotated rx 180 ry 0 rz -180 deg; joints [1.592, 71.327, -37.565, 2.864, -33.796, -2.381]
  MoveL (T13715) to (104.34, 103.54, 15.5) mm, rotated rx 180 ry 0 rz -180 deg; joints [1.395, 70.717, -36.415, 2.474, -34.326, -2.044]
  Set speed (40.0 mm/s)
  Call Extruder 2.0
  MoveL (T13716) to (104.34, 103.54, 15.5) mm, rotated rx 180 ry 0 rz -180 deg; joints [1.395, 70.717, -36.415, 2.474, -34.326, -2.044]
  Set speed (26.9 mm/s)
  MoveL (T13717) to (104.34, 103.54, 15.5) mm, rotated rx 180 ry 0 rz -180 deg; joints [1.396, 70.563, -36.125, 2.468, -34.462, -2.035]
  Call Extruder 0.0825
  MoveL (T13718) to (107.05, 103.54, 15.5) mm, rotated rx 180 ry 0 rz -180 deg; joints [1.396, 70.563, -36.125, 2.468, -34.462, -2.035]
  Call Extruder 0.05792
  MoveL (T13719) to (107.05, 105.44, 15.5) mm, rotated rx 180 ry 0 rz -180 deg; joints [1.646, 71.332, -37.573, 2.96, -33.794, -2.46]
  Call Extruder 0.11365
  MoveL (T13720) to (110.78, 105.44, 15.5) mm, rotated rx 180 ry 0 rz -180 deg; joints [1.646, 71.332, -37.573, 2.96, -33.794, -2.46]
  Call Extruder 0.05792
  MoveL (T13721) to (110.78, 103.54, 15.5) mm, rotated rx 180 ry 0 rz -180 deg; joints [1.646, 71.332, -37.573, 2.96, -33.794, -2.46]
  Call Extruder 0.0848
  MoveL (T13722) to (113.56, 103.54, 15.5) mm, rotated rx 180 ry 0 rz -180 deg; joints [1.699, 71.337, -37.582, 3.056, -33.792, -2.54]
  Call Extruder 0.05792
  MoveL (T13723) to (113.56, 105.44, 15.5) mm, rotated rx 180 ry 0 rz -180 deg; joints [1.699, 71.337, -37.582, 3.056, -33.792, -2.54]
  Call Extruder 0.11342
  MoveL (T13724) to (117.29, 105.44, 15.5) mm, rotated rx 180 ry 0 rz -180 deg; joints [1.397, 70.41, -35.838, 2.462, -34.597, -2.027]
  Call Extruder 0.05792
  MoveL (T13725) to (117.28, 103.54, 15.5) mm, rotated rx 180 ry 0 rz -180 deg; joints [1.397, 70.41, -35.838, 2.462, -34.597, -2.027]
  Call Extruder 0.12722
  MoveL (T13726) to (121.46, 103.54, 15.5) mm, rotated rx 180 ry 0 rz -180 deg; joints [1.397, 70.41, -35.838, 2.462, -34.597, -2.027]
  Call Extruder 0.09114
  MoveL (T13727) to (121.46, 106.53, 15.5) mm, rotated rx 180 ry 0 rz -180 deg; joints [1.397, 70.41, -35.838, 2.462, -34.597, -2.027]
  Call Extruder 0.05865
  MoveL (T13728) to (119.53, 106.53, 15.5) mm, rotated rx 180 ry 0 rz -180 deg; joints [1.397, 70.41, -35.838, 2.462, -34.597, -2.027]
  Call Extruder 0.11615
  MoveL (T13729) to (119.53, 110.34, 15.5) mm, rotated rx 180 ry 0 rz -180 deg; joints [1.399, 70.258, -35.552, 2.456, -34.731, -2.019]
  Call Extruder 0.05871
  MoveL (T13730) to (121.46, 110.34, 15.5) mm, rotated rx 180 ry 0 rz -180 deg; joints [1.399, 70.258, -35.552, 2.456, -34.731, -2.019]
  Call Extruder 0.10203
  MoveL (T13731) to (121.46, 113.69, 15.5) mm, rotated rx 180 ry 0 rz -180 deg; joints [1.399, 70.258, -35.552, 2.456, -34.731, -2.019]
  Call Extruder 0.05875
  MoveL (T13732) to (119.53, 113.69, 15.5) mm, rotated rx 180 ry 0 rz -180 deg; joints [1.752, 71.341, -37.591, 3.152, -33.79, -2.62]
  Call Extruder 0.11551
  MoveL (T13733) to (119.53, 117.48, 15.5) mm, rotated rx 180 ry 0 rz -180 deg; joints [1.752, 71.341, -37.591, 3.152, -33.79, -2.62]
  Call Extruder 0.0588
  MoveL (T13734) to (121.46, 117.48, 15.5) mm, rotated rx 180 ry 0 rz -180 deg; joints [1.752, 71.341, -37.591, 3.152, -33.79, -2.62]
  Call Extruder 0.12113
  MoveL (T13735) to (121.46, 121.46, 15.5) mm, rotated rx 180 ry 0 rz -180 deg; joints [1.806, 71.346, -37.6, 3.248, -33.789, -2.7]
  Call Extruder 0.54596
  MoveL (T13736) to (103.54, 121.46, 15.5) mm, rotated rx 180 ry 0 rz -180 deg; joints [1.806, 71.346, -37.6, 3.248, -33.789, -2.7]
  Call Extruder 0.54596
  MoveL (T13737) to (103.54, 103.54, 15.5) mm, rotated rx 180 ry 0 rz -180 deg; joints [1.806, 71.346, -37.6, 3.248, -33.789, -2.7]
  Call Extruder 0.02254
  MoveL (T13738) to (104.28, 103.54, 15.5) mm, rotated rx 180 ry 0 rz -180 deg; joints [1.4, 70.107, -35.267, 2.45, -34.864, -2.011]
  Set speed (150.0 mm/s)
  MoveL (T13739) to (103.53, 103.13, 15.5) mm, rotated rx 180 ry 0 rz -180 deg; joints [1.4, 70.107, -35.267, 2.45, -34.864, -2.011]
  Set speed (26.9 mm/s)
  MoveL (T13740) to (103.53, 103.13, 15.5) mm, rotated rx 180 ry 0 rz -180 deg; joints [1.401, 69.957, -34.985, 2.444, -34.996, -2.003]
  Call Extruder 0.1195
  MoveL (T13741) to (107.45, 103.13, 15.5) mm, rotated rx 180 ry 0 rz -180 deg; joints [1.401, 69.957, -34.985, 2.444, -34.996, -2.003]
  Call Extruder 0.05792
  MoveL (T13742) to (107.45, 105.03, 15.5) mm, rotated rx 180 ry 0 rz -180 deg; joints [1.401, 69.957, -34.985, 2.444, -34.996, -2.003]
  Call Extruder 0.08885
  MoveL (T13743) to (110.37, 105.03, 15.5) mm, rotated rx 180 ry 0 rz -180 deg; joints [1.859, 71.351, -37.61, 3.344, -33.787, -2.78]
  Call Extruder 0.05792
  MoveL (T13744) to (110.37, 103.13, 15.5) mm, rotated rx 180 ry 0 rz -180 deg; joints [1.859, 71.351, -37.61, 3.344, -33.787, -2.78]
  Call Extruder 0.10959
  MoveL (T13745) to (113.97, 103.13, 15.5) mm, rotated rx 180 ry 0 rz -180 deg; joints [1.859, 71.351, -37.61, 3.344, -33.787, -2.78]
  Call Extruder 0.05792
  MoveL (T13746) to (113.97, 105.03, 15.5) mm, rotated rx 180 ry 0 rz -180 deg; joints [1.912, 71.357, -37.62, 3.44, -33.785, -2.86]
  Call Extruder 0.08862
  MoveL (T13747) to (116.88, 105.03, 15.5) mm, rotated rx 180 ry 0 rz -180 deg; joints [1.912, 71.357, -37.62, 3.44, -33.785, -2.86]
  Call Extruder 0.05792
  MoveL (T13748) to (116.88, 103.13, 15.5) mm, rotated rx 180 ry 0 rz -180 deg; joints [1.912, 71.357, -37.62, 3.44, -33.785, -2.86]
  Call Extruder 0.15203
  MoveL (T13749) to (121.87, 103.13, 15.5) mm, rotated rx 180 ry 0 rz -180 deg; joints [1.912, 71.357, -37.62, 3.44, -33.785, -2.86]
  Call Extruder 0.11593
  MoveL (T13750) to (121.87, 106.94, 15.5) mm, rotated rx 180 ry 0 rz -180 deg; joints [1.403, 69.808, -34.705, 2.438, -35.127, -1.995]
  Call Extruder 0.05866
  MoveL (T13751) to (119.94, 106.94, 15.5) mm, rotated rx 180 ry 0 rz -180 deg; joints [1.403, 69.808, -34.705, 2.438, -35.127, -1.995]
  Call Extruder 0.09135
  MoveL (T13752) to (119.94, 109.94, 15.5) mm, rotated rx 180 ry 0 rz -180 deg; joints [1.404, 69.66, -34.426, 2.433, -35.258, -1.987]
  Call Extruder 0.0587
  MoveL (T13753) to (121.87, 109.94, 15.5) mm, rotated rx 180 ry 0 rz -180 deg; joints [1.404, 69.66, -34.426, 2.433, -35.258, -1.987]
  Call Extruder 0.12686
  MoveL (T13754) to (121.87, 114.1, 15.5) mm, rotated rx 180 ry 0 rz -180 deg; joints [1.966, 71.362, -37.63, 3.537, -33.783, -2.941]
  Call Extruder 0.05876
  MoveL (T13755) to (119.94, 114.1, 15.5) mm, rotated rx 180 ry 0 rz -180 deg; joints [1.966, 71.362, -37.63, 3.537, -33.783, -2.941]
  Call Extruder 0.09071
  MoveL (T13756) to (119.94, 117.08, 15.5) mm, rotated rx 180 ry 0 rz -180 deg; joints [2.019, 71.368, -37.64, 3.633, -33.78, -3.021]
  Call Extruder 0.0588
  MoveL (T13757) to (121.87, 117.08, 15.5) mm, rotated rx 180 ry 0 rz -180 deg; joints [2.019, 71.368, -37.64, 3.633, -33.78, -3.021]
  Call Extruder 0.14592
  MoveL (T13758) to (121.87, 121.87, 15.5) mm, rotated rx 180 ry 0 rz -180 deg; joints [2.019, 71.368, -37.64, 3.633, -33.78, -3.021]
  Call Extruder 0.57077
  MoveL (T13759) to (103.13, 121.87, 15.5) mm, rotated rx 180 ry 0 rz -180 deg; joints [1.405, 69.512, -34.149, 2.427, -35.388, -1.979]
  Call Extruder 0.57077
  MoveL (T13760) to (103.13, 103.13, 15.5) mm, rotated rx 180 ry 0 rz -180 deg; joints [1.405, 69.512, -34.149, 2.427, -35.388, -1.979]
  Call Extruder 0.01036
  MoveL (T13761) to (103.47, 103.13, 15.5) mm, rotated rx 180 ry 0 rz -180 deg; joints [1.405, 69.512, -34.149, 2.427, -35.388, -1.979]
  Set speed (150.0 mm/s)
  MoveL (T13762) to (102.72, 102.81, 15.5) mm, rotated rx 180 ry 0 rz -180 deg; joints [1.407, 69.366, -33.874, 2.422, -35.517, -1.972]
  Set speed (25.0 mm/s)
  MoveL (T13763) to (102.72, 102.81, 15.5) mm, rotated rx 180 ry 0 rz -180 deg; joints [1.407, 69.366, -33.874, 2.422, -35.517, -1.972]
  Call Extruder 0.00259
  MoveL (T13764) to (102.72, 102.72, 15.5) mm, rotated rx 180 ry 0 rz -180 deg; joints [2.072, 71.373, -37.651, 3.729, -33.778, -3.101]
  Call Extruder 0.15649
  MoveL (T13765) to (107.86, 102.72, 15.5) mm, rotated rx 180 ry 0 rz -180 deg; joints [2.072, 71.373, -37.651, 3.729, -33.778, -3.101]
  Call Extruder 0.05792
  MoveL (T13766) to (107.86, 104.63, 15.5) mm, rotated rx 180 ry 0 rz -180 deg; joints [2.125, 71.379, -37.662, 3.825, -33.776, -3.181]
  Call Extruder 0.06405
  MoveL (T13767) to (109.96, 104.63, 15.5) mm, rotated rx 180 ry 0 rz -180 deg; joints [2.125, 71.379, -37.662, 3.825, -33.776, -3.181]
  Call Extruder 0.05792
  MoveL (T13768) to (109.96, 102.72, 15.5) mm, rotated rx 180 ry 0 rz -180 deg; joints [1.408, 69.221, -33.6, 2.417, -35.645, -1.964]
  Call Extruder 0.13438
  MoveL (T13769) to (114.38, 102.72, 15.5) mm, rotated rx 180 ry 0 rz -180 deg; joints [1.408, 69.221, -33.6, 2.417, -35.645, -1.964]
  Call Extruder 0.05792
  MoveL (T13770) to (114.38, 104.63, 15.5) mm, rotated rx 180 ry 0 rz -180 deg; joints [1.408, 69.221, -33.6, 2.417, -35.645, -1.964]
  Call Extruder 0.06382
  MoveL (T13771) to (116.47, 104.63, 15.5) mm, rotated rx 180 ry 0 rz -180 deg; joints [1.408, 69.221, -33.6, 2.417, -35.645, -1.964]
  Call Extruder 0.05792
  MoveL (T13772) to (116.47, 102.72, 15.5) mm, rotated rx 180 ry 0 rz -180 deg; joints [1.409, 69.076, -33.328, 2.411, -35.772, -1.957]
  Call Extruder 0.17684
  MoveL (T13773) to (122.28, 102.72, 15.5) mm, rotated rx 180 ry 0 rz -180 deg; joints [1.409, 69.076, -33.328, 2.411, -35.772, -1.957]
  Call Extruder 0.14073
  MoveL (T13774) to (122.28, 107.34, 15.5) mm, rotated rx 180 ry 0 rz -180 deg; joints [1.409, 69.076, -33.328, 2.411, -35.772, -1.957]
  Call Extruder 0.05866
  MoveL (T13775) to (120.35, 107.34, 15.5) mm, rotated rx 180 ry 0 rz -180 deg; joints [2.179, 71.385, -37.673, 3.921, -33.774, -3.261]
  Call Extruder 0.06655
  MoveL (T13776) to (120.35, 109.53, 15.5) mm, rotated rx 180 ry 0 rz -180 deg; joints [2.179, 71.385, -37.673, 3.921, -33.774, -3.261]
  Call Extruder 0.05869
  MoveL (T13777) to (122.28, 109.53, 15.5) mm, rotated rx 180 ry 0 rz -180 deg; joints [2.232, 71.391, -37.685, 4.018, -33.771, -3.341]
  Call Extruder 0.15168
  MoveL (T13778) to (122.28, 114.51, 15.5) mm, rotated rx 180 ry 0 rz -180 deg; joints [2.232, 71.391, -37.685, 4.018, -33.771, -3.341]
  Call Extruder 0.05876
  MoveL (T13779) to (120.35, 114.5, 15.5) mm, rotated rx 180 ry 0 rz -180 deg; joints [2.232, 71.391, -37.685, 4.018, -33.771, -3.341]
  Call Extruder 0.06591
  MoveL (T13780) to (120.34, 116.67, 15.5) mm, rotated rx 180 ry 0 rz -180 deg; joints [2.232, 71.391, -37.685, 4.018, -33.771, -3.341]
  Call Extruder 0.05879
  MoveL (T13781) to (122.28, 116.67, 15.5) mm, rotated rx 180 ry 0 rz -180 deg; joints [1.411, 68.933, -33.058, 2.406, -35.899, -1.95]
  Call Extruder 0.1707
  MoveL (T13782) to (122.28, 122.28, 15.5) mm, rotated rx 180 ry 0 rz -180 deg; joints [1.411, 68.933, -33.058, 2.406, -35.899, -1.95]
  Call Extruder 0.59557
  MoveL (T13783) to (102.72, 122.28, 15.5) mm, rotated rx 180 ry 0 rz -180 deg; joints [1.411, 68.933, -33.058, 2.406, -35.899, -1.95]
  Call Extruder 0.59115
  MoveL (T13784) to (102.72, 102.87, 15.5) mm, rotated rx 180 ry 0 rz -180 deg; joints [1.412, 68.79, -32.789, 2.401, -36.025, -1.942]
  Set speed (150.0 mm/s)
  MoveL (T13785) to (102.78, 102.75, 15.5) mm, rotated rx 180 ry 0 rz -180 deg; joints [1.412, 68.79, -32.789, 2.401, -36.025, -1.942]
  Set speed (45.0 mm/s)
  Call Extruder -1.6
  MoveL (T13786) to (102.78, 102.75, 15.5) mm, rotated rx 180 ry 0 rz -180 deg; joints [1.412, 68.79, -32.789, 2.401, -36.025, -1.942]
  Set speed (120.0 mm/s)
  MoveL (T13787) to (102.78, 102.75, 15.5) mm, rotated rx 180 ry 0 rz -180 deg; joints [2.285, 71.397, -37.697, 4.114, -33.769, -3.422]
  Call Extruder -0.05166
  MoveL (T13788) to (102.72, 102.72, 15.5) mm, rotated rx 180 ry 0 rz -180 deg; joints [2.339, 71.404, -37.709, 4.21, -33.767, -3.502]
  Call Extruder -0.32834
  MoveL (T13789) to (103.65, 102.72, 15.5) mm, rotated rx 180 ry 0 rz -180 deg; joints [2.339, 71.404, -37.709, 4.21, -33.767, -3.502]
  Set speed (45.0 mm/s)
  Call Extruder -0.02
  MoveL (T13790) to (103.65, 102.72, 15.5) mm, rotated rx 180 ry 0 rz -180 deg; joints [1.413, 68.648, -32.522, 2.396, -36.15, -1.935]
  Set speed (150.0 mm/s)
  MoveL (T13791) to (103.65, 102.72, 17.5) mm, rotated rx 180 ry 0 rz -180 deg; joints [1.413, 68.648, -32.522, 2.396, -36.15, -1.935]
  MoveL (T13792) to (106.29, 103.84, 17.5) mm, rotated rx 180 ry 0 rz -180 deg; joints [1.413, 68.648, -32.522, 2.396, -36.15, -1.935]
  MoveL (T13793) to (106.29, 103.84, 15.5) mm, rotated rx 180 ry 0 rz -180 deg; joints [1.415, 68.506, -32.256, 2.392, -36.274, -1.928]
  Set speed (40.0 mm/s)
  Call Extruder 2.0
  MoveL (T13794) to (106.29, 103.84, 15.5) mm, rotated rx 180 ry 0 rz -180 deg; joints [1.415, 68.506, -32.256, 2.392, -36.274, -1.928]
  Set speed (26.9 mm/s)
  MoveL (T13795) to (106.29, 103.84, 15.5) mm, rotated rx 180 ry 0 rz -180 deg; joints [2.392, 71.41, -37.721, 4.306, -33.764, -3.582]
  Call Extruder 0.07441
  MoveL (T13796) to (103.84, 103.84, 15.5) mm, rotated rx 180 ry 0 rz -180 deg; joints [2.392, 71.41, -37.721, 4.306, -33.764, -3.582]
  Call Extruder 0.7458
  MoveL (T13797) to (121.16, 121.16, 15.5) mm, rotated rx 180 ry 0 rz -180 deg; joints [2.392, 71.41, -37.721, 4.306, -33.764, -3.582]
  Call Extruder 0.10254
  MoveL (T13798) to (121.16, 117.79, 15.5) mm, rotated rx 180 ry 0 rz -180 deg; joints [2.445, 71.417, -37.734, 4.403, -33.762, -3.662]
  Call Extruder 0.0039
  MoveL (T13799) to (121.03, 117.79, 15.5) mm, rotated rx 180 ry 0 rz -180 deg; joints [1.416, 68.366, -31.992, 2.387, -36.398, -1.922]
  Call Extruder 0.14502
  MoveL (T13800) to (117.66, 121.16, 15.5) mm, rotated rx 180 ry 0 rz -180 deg; joints [1.416, 68.366, -31.992, 2.387, -36.398, -1.922]
  Call Extruder 0.03385
  MoveL (T13801) to (116.55, 121.16, 15.5) mm, rotated rx 180 ry 0 rz -180 deg; joints [1.417, 68.226, -31.729, 2.382, -36.521, -1.915]
  Call Extruder 0.54738
  MoveL (T13802) to (103.84, 108.45, 15.5) mm, rotated rx 180 ry 0 rz -180 deg; joints [1.417, 68.226, -31.729, 2.382, -36.521, -1.915]
  Call Extruder 0.03385
  MoveL (T13803) to (103.84, 107.34, 15.5) mm, rotated rx 180 ry 0 rz -180 deg; joints [2.498, 71.424, -37.747, 4.499, -33.759, -3.743]
  Call Extruder 0.12482
  MoveL (T13804) to (106.74, 104.44, 15.5) mm, rotated rx 180 ry 0 rz -180 deg; joints [2.498, 71.424, -37.747, 4.499, -33.759, -3.743]
  Call Extruder 0.03972
  MoveL (T13805) to (106.74, 105.75, 15.5) mm, rotated rx 180 ry 0 rz -180 deg; joints [2.498, 71.424, -37.747, 4.499, -33.759, -3.743]
  Call Extruder 0.03468
  MoveL (T13806) to (107.88, 105.75, 15.5) mm, rotated rx 180 ry 0 rz -180 deg; joints [2.552, 71.431, -37.76, 4.595, -33.756, -3.823]
  Set speed (45.0 mm/s)
  Call Extruder -1.6
  MoveL (T13807) to (107.88, 105.75, 15.5) mm, rotated rx 180 ry 0 rz -180 deg; joints [2.552, 71.431, -37.76, 4.595, -33.756, -3.823]
  Set speed (120.0 mm/s)
  MoveL (T13808) to (107.88, 105.75, 15.5) mm, rotated rx 180 ry 0 rz -180 deg; joints [1.419, 68.087, -31.467, 2.378, -36.644, -1.908]
  Call Extruder -0.38
  MoveL (T13809) to (106.81, 105.75, 15.5) mm, rotated rx 180 ry 0 rz -180 deg; joints [1.419, 68.087, -31.467, 2.378, -36.644, -1.908]
  Set speed (45.0 mm/s)
  Call Extruder -0.02
  MoveL (T13810) to (106.81, 105.75, 15.5) mm, rotated rx 180 ry 0 rz -180 deg; joints [1.42, 67.949, -31.207, 2.373, -36.765, -1.901]
  Set speed (150.0 mm/s)
  MoveL (T13811) to (106.81, 105.75, 17.5) mm, rotated rx 180 ry 0 rz -180 deg; joints [1.42, 67.949, -31.207, 2.373, -36.765, -1.901]
  MoveL (T13812) to (110.81, 105.81, 17.5) mm, rotated rx 180 ry 0 rz -180 deg; joints [1.42, 67.949, -31.207, 2.373, -36.765, -1.901]
  MoveL (T13813) to (110.81, 105.81, 15.5) mm, rotated rx 180 ry 0 rz -180 deg; joints [2.605, 71.438, -37.773, 4.692, -33.754, -3.904]
  Set speed (40.0 mm/s)
  Call Extruder 2.0
  MoveL (T13814) to (110.81, 105.81, 15.5) mm, rotated rx 180 ry 0 rz -180 deg; joints [2.605, 71.438, -37.773, 4.692, -33.754, -3.904]
  Set speed (26.9 mm/s)
  MoveL (T13815) to (110.81, 105.81, 15.5) mm, rotated rx 180 ry 0 rz -180 deg; joints [2.658, 71.446, -37.787, 4.788, -33.751, -3.984]
  Call Extruder 0.00264
  MoveL (T13816) to (110.87, 105.87, 15.5) mm, rotated rx 180 ry 0 rz -180 deg; joints [2.658, 71.446, -37.787, 4.788, -33.751, -3.984]
  Call Extruder 0.01451
  MoveL (T13817) to (111.34, 105.87, 15.5) mm, rotated rx 180 ry 0 rz -180 deg; joints [1.421, 67.812, -30.949, 2.369, -36.886, -1.895]
  Call Extruder 0.01375
  MoveL (T13818) to (111.66, 105.55, 15.5) mm, rotated rx 180 ry 0 rz -180 deg; joints [1.421, 67.812, -30.949, 2.369, -36.886, -1.895]
  Call Extruder 0.04351
  MoveL (T13819) to (111.66, 104.13, 15.5) mm, rotated rx 180 ry 0 rz -180 deg; joints [1.423, 67.675, -30.692, 2.364, -37.007, -1.888]
  Call Extruder 0.01211
  MoveL (T13820) to (111.94, 103.84, 15.5) mm, rotated rx 180 ry 0 rz -180 deg; joints [1.423, 67.675, -30.692, 2.364, -37.007, -1.888]
  Call Extruder 0.02068
  MoveL (T13821) to (112.62, 103.84, 15.5) mm, rotated rx 180 ry 0 rz -180 deg; joints [2.711, 71.453, -37.801, 4.885, -33.748, -4.064]
  Call Extruder 0.05208
  MoveL (T13822) to (112.62, 105.55, 15.5) mm, rotated rx 180 ry 0 rz -180 deg; joints [2.711, 71.453, -37.801, 4.885, -33.748, -4.064]
  Call Extruder 0.00165
  MoveL (T13823) to (112.66, 105.59, 15.5) mm, rotated rx 180 ry 0 rz -180 deg; joints [2.765, 71.461, -37.816, 4.981, -33.745, -4.145]
  Set speed (150.0 mm/s)
  MoveL (T13824) to (112.85, 103.95, 15.5) mm, rotated rx 180 ry 0 rz -180 deg; joints [2.765, 71.461, -37.816, 4.981, -33.745, -4.145]
  Set speed (26.9 mm/s)
  MoveL (T13825) to (112.85, 103.95, 15.5) mm, rotated rx 180 ry 0 rz -180 deg; joints [2.765, 71.461, -37.816, 4.981, -33.745, -4.145]
  Call Extruder 0.01886
  MoveL (T13826) to (113.26, 104.36, 15.5) mm, rotated rx 180 ry 0 rz -180 deg; joints [1.424, 67.539, -30.436, 2.36, -37.127, -1.882]
  Call Extruder 0.02004
  MoveL (T13827) to (113.26, 104.98, 15.5) mm, rotated rx 180 ry 0 rz -180 deg; joints [1.424, 67.539, -30.436, 2.36, -37.127, -1.882]
  Call Extruder 0.01042
  MoveL (T13828) to (113.03, 104.75, 15.5) mm, rotated rx 180 ry 0 rz -180 deg; joints [1.425, 67.404, -30.181, 2.356, -37.246, -1.876]
  Call Extruder 0.02004
  MoveL (T13829) to (113.03, 105.37, 15.5) mm, rotated rx 180 ry 0 rz -180 deg; joints [2.818, 71.469, -37.83, 5.077, -33.742, -4.226]
  Call Extruder 0.01308
  MoveL (T13830) to (113.31, 105.65, 15.5) mm, rotated rx 180 ry 0 rz -180 deg; joints [2.818, 71.469, -37.83, 5.077, -33.742, -4.226]
  Set speed (45.0 mm/s)
  Call Extruder -1.6
  MoveL (T13831) to (113.31, 105.65, 15.5) mm, rotated rx 180 ry 0 rz -180 deg; joints [2.871, 71.476, -37.845, 5.174, -33.739, -4.306]
  Set speed (120.0 mm/s)
  MoveL (T13832) to (113.31, 105.65, 15.5) mm, rotated rx 180 ry 0 rz -180 deg; joints [2.871, 71.476, -37.845, 5.174, -33.739, -4.306]
  Call Extruder -0.14312
  MoveL (T13833) to (113.03, 105.37, 15.5) mm, rotated rx 180 ry 0 rz -180 deg; joints [2.871, 71.476, -37.845, 5.174, -33.739, -4.306]
  Call Extruder -0.21931
  MoveL (T13834) to (113.03, 104.75, 15.5) mm, rotated rx 180 ry 0 rz -180 deg; joints [1.427, 67.269, -29.928, 2.352, -37.364, -1.869]
  Call Extruder -0.01757
  MoveL (T13835) to (113.07, 104.78, 15.5) mm, rotated rx 180 ry 0 rz -180 deg; joints [1.428, 67.135, -29.676, 2.347, -37.482, -1.863]
  Set speed (45.0 mm/s)
  Call Extruder -0.02
  MoveL (T13836) to (113.07, 104.78, 15.5) mm, rotated rx 180 ry 0 rz -180 deg; joints [2.924, 71.485, -37.861, 5.27, -33.736, -4.387]
  Set speed (150.0 mm/s)
  MoveL (T13837) to (113.07, 104.78, 17.5) mm, rotated rx 180 ry 0 rz -180 deg; joints [2.924, 71.485, -37.861, 5.27, -33.736, -4.387]
